	!Speeds
	CONST speeddata WorkingstepSpeeddatas{140} := [
		[ 800, 500, 5000, 1000],
		[ 800, 500, 5000, 1000],
		[ 4.23333333333333, 500, 5000, 1000],
		[ 4.23333333333333, 500, 5000, 1000],
		[ 800, 500, 5000, 1000],
		[ 800, 500, 5000, 1000],
		[ 800, 500, 5000, 1000],
		[ 800, 500, 5000, 1000],
		[ 800, 500, 5000, 1000],
		[ 4.23333333333333, 500, 5000, 1000],
		[ 4.23333333333333, 500, 5000, 1000],
		[ 800, 500, 5000, 1000],
		[ 800, 500, 5000, 1000],
		[ 800, 500, 5000, 1000],
		[ 800, 500, 5000, 1000],
		[ 800, 500, 5000, 1000],
		[ 4.23333333333333, 500, 5000, 1000],
		[ 4.23333333333333, 500, 5000, 1000],
		[ 800, 500, 5000, 1000],
		[ 800, 500, 5000, 1000],
		[ 800, 500, 5000, 1000],
		[ 800, 500, 5000, 1000],
		[ 800, 500, 5000, 1000],
		[ 4.23333333333333, 500, 5000, 1000],
		[ 4.23333333333333, 500, 5000, 1000],
		[ 800, 500, 5000, 1000],
		[ 800, 500, 5000, 1000],
		[ 800, 500, 5000, 1000],
		[ 800, 500, 5000, 1000],
		[ 800, 500, 5000, 1000],
		[ 4.23333333333333, 500, 5000, 1000],
		[ 4.23333333333333, 500, 5000, 1000],
		[ 800, 500, 5000, 1000],
		[ 800, 500, 5000, 1000],
		[ 800, 500, 5000, 1000],
		[ 800, 500, 5000, 1000],
		[ 800, 500, 5000, 1000],
		[ 4.23333333333333, 500, 5000, 1000],
		[ 4.23333333333333, 500, 5000, 1000],
		[ 800, 500, 5000, 1000],
		[ 800, 500, 5000, 1000],
		[ 800, 500, 5000, 1000],
		[ 800, 500, 5000, 1000],
		[ 800, 500, 5000, 1000],
		[ 4.23333333333333, 500, 5000, 1000],
		[ 4.23333333333333, 500, 5000, 1000],
		[ 800, 500, 5000, 1000],
		[ 800, 500, 5000, 1000],
		[ 800, 500, 5000, 1000],
		[ 800, 500, 5000, 1000],
		[ 800, 500, 5000, 1000],
		[ 4.23333333333333, 500, 5000, 1000],
		[ 4.23333333333333, 500, 5000, 1000],
		[ 800, 500, 5000, 1000],
		[ 800, 500, 5000, 1000],
		[ 800, 500, 5000, 1000],
		[ 800, 500, 5000, 1000],
		[ 800, 500, 5000, 1000],
		[ 4.23333333333333, 500, 5000, 1000],
		[ 4.23333333333333, 500, 5000, 1000],
		[ 800, 500, 5000, 1000],
		[ 800, 500, 5000, 1000],
		[ 800, 500, 5000, 1000],
		[ 800, 500, 5000, 1000],
		[ 800, 500, 5000, 1000],
		[ 4.23333333333333, 500, 5000, 1000],
		[ 4.23333333333333, 500, 5000, 1000],
		[ 800, 500, 5000, 1000],
		[ 800, 500, 5000, 1000],
		[ 800, 500, 5000, 1000],
		[ 800, 500, 5000, 1000],
		[ 800, 500, 5000, 1000],
		[ 4.23333333333333, 500, 5000, 1000],
		[ 4.23333333333333, 500, 5000, 1000],
		[ 800, 500, 5000, 1000],
		[ 800, 500, 5000, 1000],
		[ 800, 500, 5000, 1000],
		[ 800, 500, 5000, 1000],
		[ 800, 500, 5000, 1000],
		[ 4.23333333333333, 500, 5000, 1000],
		[ 4.23333333333333, 500, 5000, 1000],
		[ 800, 500, 5000, 1000],
		[ 800, 500, 5000, 1000],
		[ 800, 500, 5000, 1000],
		[ 800, 500, 5000, 1000],
		[ 800, 500, 5000, 1000],
		[ 4.23333333333333, 500, 5000, 1000],
		[ 4.23333333333333, 500, 5000, 1000],
		[ 800, 500, 5000, 1000],
		[ 800, 500, 5000, 1000],
		[ 800, 500, 5000, 1000],
		[ 800, 500, 5000, 1000],
		[ 800, 500, 5000, 1000],
		[ 4.23333333333333, 500, 5000, 1000],
		[ 4.23333333333333, 500, 5000, 1000],
		[ 800, 500, 5000, 1000],
		[ 800, 500, 5000, 1000],
		[ 800, 500, 5000, 1000],
		[ 800, 500, 5000, 1000],
		[ 800, 500, 5000, 1000],
		[ 4.23333333333333, 500, 5000, 1000],
		[ 4.23333333333333, 500, 5000, 1000],
		[ 800, 500, 5000, 1000],
		[ 800, 500, 5000, 1000],
		[ 800, 500, 5000, 1000],
		[ 800, 500, 5000, 1000],
		[ 800, 500, 5000, 1000],
		[ 4.23333333333333, 500, 5000, 1000],
		[ 4.23333333333333, 500, 5000, 1000],
		[ 800, 500, 5000, 1000],
		[ 800, 500, 5000, 1000],
		[ 800, 500, 5000, 1000],
		[ 800, 500, 5000, 1000],
		[ 800, 500, 5000, 1000],
		[ 4.23333333333333, 500, 5000, 1000],
		[ 4.23333333333333, 500, 5000, 1000],
		[ 800, 500, 5000, 1000],
		[ 800, 500, 5000, 1000],
		[ 800, 500, 5000, 1000],
		[ 800, 500, 5000, 1000],
		[ 800, 500, 5000, 1000],
		[ 4.23333333333333, 500, 5000, 1000],
		[ 4.23333333333333, 500, 5000, 1000],
		[ 800, 500, 5000, 1000],
		[ 800, 500, 5000, 1000],
		[ 800, 500, 5000, 1000],
		[ 800, 500, 5000, 1000],
		[ 800, 500, 5000, 1000],
		[ 4.23333333333333, 500, 5000, 1000],
		[ 4.23333333333333, 500, 5000, 1000],
		[ 800, 500, 5000, 1000],
		[ 800, 500, 5000, 1000],
		[ 800, 500, 5000, 1000],
		[ 800, 500, 5000, 1000],
		[ 800, 500, 5000, 1000],
		[ 4.23333333333333, 500, 5000, 1000],
		[ 4.23333333333333, 500, 5000, 1000],
		[ 800, 500, 5000, 1000],
		[ 800, 500, 5000, 1000],
		[ 800, 500, 5000, 1000]
		];


ENDMODULE

--- Backups/Rob2/RAPID/TASK1/PROGMOD/KyleWorkingPlan.mod ---
MODULE KyleWorkingPlan
  PERS string workingPlanUUID:="sdvonvskvnwovewn342532nkfloencvosnvqwef12";
    PERS string AP238_WORKINGSTEP_NAME := "";
    PERS string AP238_WORKINGSTEP_UUID := "";
    PERS string AP238_FEATURE_NAME := "";
    PERS string AP238_FEATURE_UUID := "";
    PERS bool ok;
    PERS num startIndex :=134;
    PERS num stopIndex :=140;
      CONST speeddata serge := [ 800, 500, 5000, 1000];



    PROC main()

       !  SetDO IsDone,0;
         MoveAbsJ jHome,v400,z10,PendEff_point\WObj:=A;
        MoveAbsJ jee,v400,z10,PendEff_point\WObj:=A;
        ConfJ\Off;
        ConfL\Off;

       FOR i FROM 1 TO dim(WorkPlan,1) DO

           ok := StrToVal(Workplan{i,1}, startIndex);
           ok := StrToVal(Workplan{i,2}, stopIndex);

                WorkingStep startIndex, stopIndex, Workplan{i,3}, Workplan{i,4}, Workplan{i,5}, Workplan{i,6}, WorkingstepRobtargets, WorkingstepSpeeddatas;

        ENDFOR

        MoveAbsJ jee,v400,z10,PendEff_point\WObj:=A;
        MoveAbsJ jHome,v400,z10,PendEff_point\WObj:=A;
        !SetDO IsDone,0;
    ENDPROC

    PROC WorkingStep(num startpos, num endpos, string workingstepName, string workingstepUUID, string featureName, string featureUUID, robtarget targetList{*}, speeddata speedList{*})

        FOR i FROM startpos TO endpos DO
      !           SetDO IsDone,0;
            AP238_WORKINGSTEP_NAME := workingstepName;
            AP238_WORKINGSTEP_UUID := workingstepUUID;
            AP238_FEATURE_NAME := featureName;
            AP238_FEATURE_UUID := featureUUID;
     !       MoveL targetList{i},v1000,z100,PendEff_point\WObj:=A;
            MoveL Workingsteprobtargets{i}, speedList{i}, z100,PendEff_point\WObj:=A;
     !       SetDO IsDone,1;
            AP238_WORKINGSTEP_NAME := "";
            AP238_WORKINGSTEP_UUID := "";
            AP238_FEATURE_NAME := "";
            AP238_FEATURE_UUID := "";
        ENDFOR

    ENDPROC

ENDMODULE

--- Backups/Rob2/RAPID/TASK1/SYSMOD/StandardJointMoves.sys ---
MODULE StandardJointMoves(SYSMODULE)
    !Home Joint Target
    CONST jointtarget jHome:=[[0,0,0,0,0,0],[9E+09,9E+09,9E+09,9E+09,9E+09,9E+09]];
    !Entry/Exit Joint Targets
    CONST jointtarget jee:=[[90,14,18,4,-38,0],[9E+09,9E+09,9E+09,9E+09,9E+09,9E+09]];
ENDMODULE

--- Backups/Rob2/RAPID/TASK1/SYSMOD/WorkObjs.sys ---
MODULE WorkObjs(SYSMODULE)
   TASK PERS wobjdata A:=[FALSE,TRUE,"",[[246.014,597.3,290.101],[0,0,0,1]],[[0,0,0],[1,0,0,0]]];
ENDMODULE

--- Backups/Rob3/RAPID/TASK1/PROGMOD/CartmanTargets.mod ---
MODULE CartmanTargets

	!Workplan Variables
	CONST string workplanName := "Cartman";
	CONST string workplanUUID := "e8924aac-08a1-45c9-8646-5367342a41b0";

	!Workingsteps
	CONST string WorkPlan{20,6} := [
		["1","7", "Drilling.82", "d2e6eab3-8d0a-4f0f-a95d-911cd3530854", "Hole.182", "99ddfef0-3deb-445b-9c3c-e9123ea0c45e"],
		["8","14", "Drilling.77", "18dec0f3-9a71-4d62-9ffd-4b071a4c2c96", "Hole.187", "ac14d56a-bac8-4703-abe8-8083d949a042"],
		["15","21", "Drilling.77A", "cce52ede-30b0-41b1-9812-f49428268d42", "Hole.186", "13f6412f-3d62-4080-9683-c1b012cf2329"],
		["22","28", "Drilling.81", "cc8ebbb7-3856-4b1d-89e7-3bb7927c75a5", "Hole.183", "cc7cadc1-0fbf-4952-a172-cb43c9784d58"],
		["29","35", "Drilling.82A", "fb1fd053-2caa-42bb-a221-a69a247b4566", "Hole.181", "d6ab53ed-32cb-4e94-b962-5e5bce2dd949"],
		["36","42", "Drilling.78", "0ce5bf9a-dc56-429d-9ede-9ff3cf936782", "Hole.188", "61b61ac0-b937-4570-af27-f3e5565ecb41"],
		["43","49", "Drilling.80", "097974f7-0281-41d6-be47-a718a708f2c1", "Hole.184", "41873095-e461-4717-85b4-deda62e7cc48"],
		["50","56", "Drilling.79", "0d38a1e5-c414-47eb-bffd-0c035c73e724", "Hole.189", "7aab888b-ee1b-4aa6-95a1-195311f5c09c"],
		["57","63", "Drilling.56", "71fb19fa-6caa-4311-b6e3-cc7c1a002d0e", "Hole.193", "534c8ca5-8759-4bfe-8b3a-f64014fb1b37"],
		["64","70", "Drilling.57", "82dc275d-79a1-4817-aca9-f89dbea4337b", "Hole.194", "b7011f38-5032-4673-a101-1254335b2b68"],
		["71","77", "Drilling.58", "e8ffa874-f10e-4ad9-b179-7e628cd38fb4", "Hole.195", "b2305f3a-4977-4727-8945-7fbced9dd981"],
		["78","84", "Drilling.59", "0436a6f4-bfce-4d24-b9fc-4974d9771220", "Hole.196", "3f2baa8f-1c3f-4c1c-9c8e-c6857731bbd6"],
		["85","91", "Drilling.60", "c922b515-5149-48e0-b3c2-25974a63925d", "Hole.199", "9f4fe053-f702-4970-bd3b-e9d6d5939926"],
		["92","98", "Drilling.61", "54f7aa6c-4c3b-4a01-975b-a374c0101e01", "Hole.198", "0cbf5231-fc2b-4c71-8eca-d485859f5bef"],
		["99","105", "Drilling.62", "308c7519-319c-495b-866e-887c108f69fd", "Hole.197", "97270ee4-7d12-42d9-b2be-af7000f13095"],
		["106","112", "Drilling.63", "ae041463-52c1-413a-bc8f-b82ceccd6cbf", "Hole.192", "a8675cfd-087c-4d76-9144-1d9942c5b76b"],
		["113","119", "Drilling.96", "366ca4c1-51ca-4762-a30e-71a9ecae8757", "Hole.176", "5d7c72e5-ba80-4f5c-9be4-85262b61495c"],
		["120","126", "Drilling.97", "81b03597-23b4-45f9-8253-620e9a46ff2e", "Hole.177", "fbc5cc65-6031-4a9a-8bf6-0c8b0c46d944"],
		["127","133", "Drilling.98", "d04a2e7a-5080-477a-8967-be3c7ad103b0", "Hole.178", "14004e87-3834-406b-b1c2-5711ea87ae56"],
		["134","140", "Drilling.99", "80c84945-9521-4e27-bda3-a7734aa46377", "Hole.179", "ec45e44e-466b-44fe-87e7-d5d7371b5502"]
		];

	!Positions
	CONST robtarget WorkingstepRobtargets{140} := [
		[[1250.47999638542,-108.227438181067,34.9975797061398],[0.00721600922388558,-0.000419915796535777,-0.998285039502953,-0.0580924503373097],[0,0,0,0],[9E+09,9E+09,9E+09,9E+09,9E+09,9E+09]],
		[[1249.75058558968,-102.335059394747,-15.4542570506085],[0.00721600922388558,-0.000419915796535777,-0.998285039502953,-0.0580924503373097],[0,0,0,0],[9E+09,9E+09,9E+09,9E+09,9E+09,9E+09]],
		[[1249.75058558968,-102.335059394747,-15.4542570506085],[0.00721600922388558,-0.000419915796535777,-0.998285039502953,-0.0580924503373097],[0,0,0,0],[9E+09,9E+09,9E+09,9E+09,9E+09,9E+09]],
		[[1249.29470384234,-98.6523226532974,-46.9866550235762],[0.00721600922388558,-0.000419915796535777,-0.998285039502953,-0.0580924503373097],[0,0,0,0],[9E+09,9E+09,9E+09,9E+09,9E+09,9E+09]],
		[[1249.29470384234,-98.6523226532974,-46.9866550235762],[0.00721600922388558,-0.000419915796535777,-0.998285039502953,-0.0580924503373097],[0,0,0,0],[9E+09,9E+09,9E+09,9E+09,9E+09,9E+09]],
		[[1249.75058558968,-102.335059394747,-15.4542570506085],[0.00721600922388558,-0.000419915796535777,-0.998285039502953,-0.0580924503373097],[0,0,0,0],[9E+09,9E+09,9E+09,9E+09,9E+09,9E+09]],
		[[1250.47999638542,-108.227438181067,34.9975797061398],[0.00721600922388558,-0.000419915796535777,-0.998285039502953,-0.0580924503373097],[0,0,0,0],[9E+09,9E+09,9E+09,9E+09,9E+09,9E+09]],
		[[1190.4996392186,-113.751032090431,35.2122877951345],[0.00727717079532053,-0.000437833858996109,-0.998168434785264,-0.0600551986514469],[0,0,0,0],[9E+09,9E+09,9E+09,9E+09,9E+09,9E+09]],
		[[1189.76430434352,-107.660275683661,-15.2158984603209],[0.00727717079532053,-0.000437833858996109,-0.998168434785264,-0.0600551986514469],[0,0,0,0],[9E+09,9E+09,9E+09,9E+09,9E+09,9E+09]],
		[[1189.76430434352,-107.660275683661,-15.2158984603209],[0.00727717079532053,-0.000437833858996109,-0.998168434785264,-0.0600551986514469],[0,0,0,0],[9E+09,9E+09,9E+09,9E+09,9E+09,9E+09]],
		[[1189.3047200466,-103.853552929431,-46.7335148699807],[0.00727717079532053,-0.000437833858996109,-0.998168434785264,-0.0600551986514469],[0,0,0,0],[9E+09,9E+09,9E+09,9E+09,9E+09,9E+09]],
		[[1189.3047200466,-103.853552929431,-46.7335148699807],[0.00727717079532053,-0.000437833858996109,-0.998168434785264,-0.0600551986514469],[0,0,0,0],[9E+09,9E+09,9E+09,9E+09,9E+09,9E+09]],
		[[1189.76430434352,-107.660275683661,-15.2158984603209],[0.00727717079532053,-0.000437833858996109,-0.998168434785264,-0.0600551986514469],[0,0,0,0],[9E+09,9E+09,9E+09,9E+09,9E+09,9E+09]],
		[[1190.4996392186,-113.751032090431,35.2122877951345],[0.00727717079532053,-0.000437833858996109,-0.998168434785264,-0.0600551986514469],[0,0,0,0],[9E+09,9E+09,9E+09,9E+09,9E+09,9E+09]],
		[[1189.80854349765,-65.9236756789968,39.7730886825223],[0.00665335945126355,-0.000231418506074151,-0.999373500218657,-0.0347604130326124],[0,0,0,0],[9E+09,9E+09,9E+09,9E+09,9E+09,9E+09]],
		[[1189.13380297056,-62.3940738632379,-10.8996518812492],[0.00665335945126355,-0.000231418506074151,-0.999373500218657,-0.0347604130326124],[0,0,0,0],[9E+09,9E+09,9E+09,9E+09,9E+09,9E+09]],
		[[1189.13380297056,-62.3940738632379,-10.8996518812492],[0.00665335945126355,-0.000231418506074151,-0.999373500218657,-0.0347604130326124],[0,0,0,0],[9E+09,9E+09,9E+09,9E+09,9E+09,9E+09]],
		[[1188.71209014113,-60.1880727283885,-42.5701147336066],[0.00665335945126355,-0.000231418506074151,-0.999373500218657,-0.0347604130326124],[0,0,0,0],[9E+09,9E+09,9E+09,9E+09,9E+09,9E+09]],
		[[1188.71209014113,-60.1880727283885,-42.5701147336066],[0.00665335945126355,-0.000231418506074151,-0.999373500218657,-0.0347604130326124],[0,0,0,0],[9E+09,9E+09,9E+09,9E+09,9E+09,9E+09]],
		[[1189.13380297056,-62.3940738632379,-10.8996518812492],[0.00665335945126355,-0.000231418506074151,-0.999373500218657,-0.0347604130326124],[0,0,0,0],[9E+09,9E+09,9E+09,9E+09,9E+09,9E+09]],
		[[1189.80854349765,-65.9236756789968,39.7730886825223],[0.00665335945126355,-0.000231418506074151,-0.999373500218657,-0.0347604130326124],[0,0,0,0],[9E+09,9E+09,9E+09,9E+09,9E+09,9E+09]],
		[[1251.74376412468,-153.597058265429,28.5448951127816],[0.00812040995990566,-0.000673216620954281,-0.996547971260864,-0.0826180773034575],[0,0,0,0],[9E+09,9E+09,9E+09,9E+09,9E+09,9E+09]],
		[[1250.92722949069,-145.231482502716,-21.5549094112862],[0.00812040995990566,-0.000673216620954281,-0.996547971260864,-0.0826180773034575],[0,0,0,0],[9E+09,9E+09,9E+09,9E+09,9E+09,9E+09]],
		[[1250.92722949069,-145.231482502716,-21.5549094112862],[0.00812040995990566,-0.000673216620954281,-0.996547971260864,-0.0826180773034575],[0,0,0,0],[9E+09,9E+09,9E+09,9E+09,9E+09,9E+09]],
		[[1250.41689534445,-140.002997651021,-52.8672872388287],[0.00812040995990566,-0.000673216620954281,-0.996547971260864,-0.0826180773034575],[0,0,0,0],[9E+09,9E+09,9E+09,9E+09,9E+09,9E+09]],
		[[1250.41689534445,-140.002997651021,-52.8672872388287],[0.00812040995990566,-0.000673216620954281,-0.996547971260864,-0.0826180773034575],[0,0,0,0],[9E+09,9E+09,9E+09,9E+09,9E+09,9E+09]],
		[[1250.92722949069,-145.231482502716,-21.5549094112862],[0.00812040995990566,-0.000673216620954281,-0.996547971260864,-0.0826180773034575],[0,0,0,0],[9E+09,9E+09,9E+09,9E+09,9E+09,9E+09]],
		[[1251.74376412468,-153.597058265429,28.5448951127816],[0.00812040995990566,-0.000673216620954281,-0.996547971260864,-0.0826180773034575],[0,0,0,0],[9E+09,9E+09,9E+09,9E+09,9E+09,9E+09]],
		[[1251.30388547251,-68.6381103493351,38.7572467507825],[0.0066912868110706,-0.000246540181525224,-0.99929951275717,-0.0368191485783281],[0,0,0,0],[9E+09,9E+09,9E+09,9E+09,9E+09,9E+09]],
		[[1250.62544921187,-64.8997376477342,-11.9004702702614],[0.0066912868110706,-0.000246540181525224,-0.99929951275717,-0.0368191485783281],[0,0,0,0],[9E+09,9E+09,9E+09,9E+09,9E+09,9E+09]],
		[[1250.62544921187,-64.8997376477342,-11.9004702702614],[0.0066912868110706,-0.000246540181525224,-0.99929951275717,-0.0368191485783281],[0,0,0,0],[9E+09,9E+09,9E+09,9E+09,9E+09,9E+09]],
		[[1250.20142654896,-62.5632547092337,-43.5615434084138],[0.0066912868110706,-0.000246540181525224,-0.99929951275717,-0.0368191485783281],[0,0,0,0],[9E+09,9E+09,9E+09,9E+09,9E+09,9E+09]],
		[[1250.20142654896,-62.5632547092337,-43.5615434084138],[0.0066912868110706,-0.000246540181525224,-0.99929951275717,-0.0368191485783281],[0,0,0,0],[9E+09,9E+09,9E+09,9E+09,9E+09,9E+09]],
		[[1250.62544921187,-64.8997376477342,-11.9004702702614],[0.0066912868110706,-0.000246540181525224,-0.99929951275717,-0.0368191485783281],[0,0,0,0],[9E+09,9E+09,9E+09,9E+09,9E+09,9E+09]],
		[[1251.30388547251,-68.6381103493351,38.7572467507825],[0.0066912868110706,-0.000246540181525224,-0.99929951275717,-0.0368191485783281],[0,0,0,0],[9E+09,9E+09,9E+09,9E+09,9E+09,9E+09]],
		[[1190.60083196625,-155.158216713176,29.2801865539037],[0.00809702025081855,-0.000666620341839099,-0.996595199463999,-0.0820487799159123],[0,0,0,0],[9E+09,9E+09,9E+09,9E+09,9E+09,9E+09]],
		[[1189.78653274383,-146.849895222209,-20.8291809413968],[0.00809702025081855,-0.000666620341839099,-0.996595199463999,-0.0820487799159123],[0,0,0,0],[9E+09,9E+09,9E+09,9E+09,9E+09,9E+09]],
		[[1189.78653274383,-146.849895222209,-20.8291809413968],[0.00809702025081855,-0.000666620341839099,-0.996595199463999,-0.0820487799159123],[0,0,0,0],[9E+09,9E+09,9E+09,9E+09,9E+09,9E+09]],
		[[1189.27759572982,-141.657194290354,-52.1475356259597],[0.00809702025081855,-0.000666620341839099,-0.996595199463999,-0.0820487799159123],[0,0,0,0],[9E+09,9E+09,9E+09,9E+09,9E+09,9E+09]],
		[[1189.27759572982,-141.657194290354,-52.1475356259597],[0.00809702025081855,-0.000666620341839099,-0.996595199463999,-0.0820487799159123],[0,0,0,0],[9E+09,9E+09,9E+09,9E+09,9E+09,9E+09]],
		[[1189.78653274383,-146.849895222209,-20.8291809413968],[0.00809702025081855,-0.000666620341839099,-0.996595199463999,-0.0820487799159123],[0,0,0,0],[9E+09,9E+09,9E+09,9E+09,9E+09,9E+09]],
		[[1190.60083196625,-155.158216713176,29.2801865539037],[0.00809702025081855,-0.000666620341839099,-0.996595199463999,-0.0820487799159123],[0,0,0,0],[9E+09,9E+09,9E+09,9E+09,9E+09,9E+09]],
		[[1251.64830610495,-198.940144194599,19.8167872449908],[0.00936178502431022,-0.00100991908065343,-0.99418752340432,-0.107249733574467],[0,0,0,0],[9E+09,9E+09,9E+09,9E+09,9E+09,9E+09]],
		[[1250.71368198328,-188.105946746604,-29.8056536805528],[0.00936178502431022,-0.00100991908065343,-0.99418752340432,-0.107249733574467],[0,0,0,0],[9E+09,9E+09,9E+09,9E+09,9E+09,9E+09]],
		[[1250.71368198328,-188.105946746604,-29.8056536805528],[0.00936178502431022,-0.00100991908065343,-0.99418752340432,-0.107249733574467],[0,0,0,0],[9E+09,9E+09,9E+09,9E+09,9E+09,9E+09]],
		[[1250.12954190724,-181.334573341607,-60.8196792590172],[0.00936178502431022,-0.00100991908065343,-0.99418752340432,-0.107249733574467],[0,0,0,0],[9E+09,9E+09,9E+09,9E+09,9E+09,9E+09]],
		[[1250.12954190724,-181.334573341607,-60.8196792590172],[0.00936178502431022,-0.00100991908065343,-0.99418752340432,-0.107249733574467],[0,0,0,0],[9E+09,9E+09,9E+09,9E+09,9E+09,9E+09]],
		[[1250.71368198328,-188.105946746604,-29.8056536805528],[0.00936178502431022,-0.00100991908065343,-0.99418752340432,-0.107249733574467],[0,0,0,0],[9E+09,9E+09,9E+09,9E+09,9E+09,9E+09]],
		[[1251.64830610495,-198.940144194599,19.8167872449908],[0.00936178502431022,-0.00100991908065343,-0.99418752340432,-0.107249733574467],[0,0,0,0],[9E+09,9E+09,9E+09,9E+09,9E+09,9E+09]],
		[[1191.95221981654,-205.961103975954,19.400651812078],[0.00947883770226787,-0.00104166552827841,-0.99397062768479,-0.109231212886453],[0,0,0,0],[9E+09,9E+09,9E+09,9E+09,9E+09,9E+09]],
		[[1191.00653678319,-194.929122888932,-30.1779834746662],[0.00947883770226787,-0.00104166552827841,-0.99397062768479,-0.109231212886453],[0,0,0,0],[9E+09,9E+09,9E+09,9E+09,9E+09,9E+09]],
		[[1191.00653678319,-194.929122888932,-30.1779834746662],[0.00947883770226787,-0.00104166552827841,-0.99397062768479,-0.109231212886453],[0,0,0,0],[9E+09,9E+09,9E+09,9E+09,9E+09,9E+09]],
		[[1190.41548488734,-188.034134709543,-61.1646305288814],[0.00947883770226787,-0.00104166552827841,-0.99397062768479,-0.109231212886453],[0,0,0,0],[9E+09,9E+09,9E+09,9E+09,9E+09,9E+09]],
		[[1190.41548488734,-188.034134709543,-61.1646305288814],[0.00947883770226787,-0.00104166552827841,-0.99397062768479,-0.109231212886453],[0,0,0,0],[9E+09,9E+09,9E+09,9E+09,9E+09,9E+09]],
		[[1191.00653678319,-194.929122888932,-30.1779834746662],[0.00947883770226787,-0.00104166552827841,-0.99397062768479,-0.109231212886453],[0,0,0,0],[9E+09,9E+09,9E+09,9E+09,9E+09,9E+09]],
		[[1191.95221981654,-205.961103975954,19.400651812078],[0.00947883770226787,-0.00104166552827841,-0.99397062768479,-0.109231212886453],[0,0,0,0],[9E+09,9E+09,9E+09,9E+09,9E+09,9E+09]],
		[[1047.46148935396,-72.0531501973382,41.2352412437369],[0.00668721181442413,-0.000244662737514811,-0.999309004762805,-0.0365613776855514],[0,0,0,0],[9E+09,9E+09,9E+09,9E+09,9E+09,9E+09]],
		[[1046.7834469431,-68.3409147913177,-9.42440311722726],[0.00668721181442413,-0.000244662737514811,-0.999309004762805,-0.0365613776855514],[0,0,0,0],[9E+09,9E+09,9E+09,9E+09,9E+09,9E+09]],
		[[1046.7834469431,-68.3409147913177,-9.42440311722726],[0.00668721181442413,-0.000244662737514811,-0.999309004762805,-0.0365613776855514],[0,0,0,0],[9E+09,9E+09,9E+09,9E+09,9E+09,9E+09]],
		[[1046.35967043631,-66.0207676625549,-41.0866808428298],[0.00668721181442413,-0.000244662737514811,-0.999309004762805,-0.0365613776855514],[0,0,0,0],[9E+09,9E+09,9E+09,9E+09,9E+09,9E+09]],
		[[1046.35967043631,-66.0207676625549,-41.0866808428298],[0.00668721181442413,-0.000244662737514811,-0.999309004762805,-0.0365613776855514],[0,0,0,0],[9E+09,9E+09,9E+09,9E+09,9E+09,9E+09]],
		[[1046.7834469431,-68.3409147913177,-9.42440311722726],[0.00668721181442413,-0.000244662737514811,-0.999309004762805,-0.0365613776855514],[0,0,0,0],[9E+09,9E+09,9E+09,9E+09,9E+09,9E+09]],
		[[1047.46148935396,-72.0531501973382,41.2352412437369],[0.00668721181442413,-0.000244662737514811,-0.999309004762805,-0.0365613776855514],[0,0,0,0],[9E+09,9E+09,9E+09,9E+09,9E+09,9E+09]],
		[[1052.42343074024,-109.067908351377,37.7494232893189],[0.00713988796543304,-0.000396579657530434,-0.998435450217324,-0.0554573392234659],[0,0,0,0],[9E+09,9E+09,9E+09,9E+09,9E+09,9E+09]],
		[[1051.70138758157,-103.441970404417,-12.7329248721323],[0.00713988796543304,-0.000396579657530434,-0.998435450217324,-0.0554573392234659],[0,0,0,0],[9E+09,9E+09,9E+09,9E+09,9E+09,9E+09]],
		[[1051.70138758157,-103.441970404417,-12.7329248721323],[0.00713988796543304,-0.000396579657530434,-0.998435450217324,-0.0554573392234659],[0,0,0,0],[9E+09,9E+09,9E+09,9E+09,9E+09,9E+09]],
		[[1051.2501106074,-99.9257591875673,-44.2843924730394],[0.00713988796543304,-0.000396579657530434,-0.998435450217324,-0.0554573392234659],[0,0,0,0],[9E+09,9E+09,9E+09,9E+09,9E+09,9E+09]],
		[[1051.2501106074,-99.9257591875673,-44.2843924730394],[0.00713988796543304,-0.000396579657530434,-0.998435450217324,-0.0554573392234659],[0,0,0,0],[9E+09,9E+09,9E+09,9E+09,9E+09,9E+09]],
		[[1051.70138758157,-103.441970404417,-12.7329248721323],[0.00713988796543304,-0.000396579657530434,-0.998435450217324,-0.0554573392234659],[0,0,0,0],[9E+09,9E+09,9E+09,9E+09,9E+09,9E+09]],
		[[1052.42343074024,-109.067908351377,37.7494232893189],[0.00713988796543304,-0.000396579657530434,-0.998435450217324,-0.0554573392234659],[0,0,0,0],[9E+09,9E+09,9E+09,9E+09,9E+09,9E+09]],
		[[1058.4740893206,-161.105031430509,30.4416121484464],[0.00810621924312884,-0.000668612028545384,-0.996582703082117,-0.0821995017325489],[0,0,0,0],[9E+09,9E+09,9E+09,9E+09,9E+09,9E+09]],
		[[1057.65889579635,-152.781550841607,-19.6652250138031],[0.00810621924312884,-0.000668612028545384,-0.996582703082117,-0.0821995017325489],[0,0,0,0],[9E+09,9E+09,9E+09,9E+09,9E+09,9E+09]],
		[[1057.65889579635,-152.781550841607,-19.6652250138031],[0.00810621924312884,-0.000668612028545384,-0.996582703082117,-0.0821995017325489],[0,0,0,0],[9E+09,9E+09,9E+09,9E+09,9E+09,9E+09]],
		[[1057.1493998437,-147.579375473542,-50.981998240209],[0.00810621924312884,-0.000668612028545384,-0.996582703082117,-0.0821995017325489],[0,0,0,0],[9E+09,9E+09,9E+09,9E+09,9E+09,9E+09]],
		[[1057.1493998437,-147.579375473542,-50.981998240209],[0.00810621924312884,-0.000668612028545384,-0.996582703082117,-0.0821995017325489],[0,0,0,0],[9E+09,9E+09,9E+09,9E+09,9E+09,9E+09]],
		[[1057.65889579635,-152.781550841607,-19.6652250138031],[0.00810621924312884,-0.000668612028545384,-0.996582703082117,-0.0821995017325489],[0,0,0,0],[9E+09,9E+09,9E+09,9E+09,9E+09,9E+09]],
		[[1058.4740893206,-161.105031430509,30.4416121484464],[0.00810621924312884,-0.000668612028545384,-0.996582703082117,-0.0821995017325489],[0,0,0,0],[9E+09,9E+09,9E+09,9E+09,9E+09,9E+09]],
		[[1057.93506911126,-221.171435306608,18.5414921384049],[0.00971864696644204,-0.00110695702979796,-0.993528265759436,-0.113163190500817],[0,0,0,0],[9E+09,9E+09,9E+09,9E+09,9E+09,9E+09]],
		[[1056.96677196969,-209.747370115093,-30.9478313076238],[0.00971864696644204,-0.00110695702979796,-0.993528265759436,-0.113163190500817],[0,0,0,0],[9E+09,9E+09,9E+09,9E+09,9E+09,9E+09]],
		[[1056.96677196969,-209.747370115093,-30.9478313076238],[0.00971864696644204,-0.00110695702979796,-0.993528265759436,-0.113163190500817],[0,0,0,0],[9E+09,9E+09,9E+09,9E+09,9E+09,9E+09]],
		[[1056.36158625621,-202.607329370396,-61.8786584613916],[0.00971864696644204,-0.00110695702979796,-0.993528265759436,-0.113163190500817],[0,0,0,0],[9E+09,9E+09,9E+09,9E+09,9E+09,9E+09]],
		[[1056.36158625621,-202.607329370396,-61.8786584613916],[0.00971864696644204,-0.00110695702979796,-0.993528265759436,-0.113163190500817],[0,0,0,0],[9E+09,9E+09,9E+09,9E+09,9E+09,9E+09]],
		[[1056.96677196969,-209.747370115093,-30.9478313076238],[0.00971864696644204,-0.00110695702979796,-0.993528265759436,-0.113163190500817],[0,0,0,0],[9E+09,9E+09,9E+09,9E+09,9E+09,9E+09]],
		[[1057.93506911126,-221.171435306608,18.5414921384049],[0.00971864696644204,-0.00110695702979796,-0.993528265759436,-0.113163190500817],[0,0,0,0],[9E+09,9E+09,9E+09,9E+09,9E+09,9E+09]],
		[[1127.85981856446,-218.635862664587,17.7574554971789],[0.00976696523800443,-0.0011207663604795,-0.993432439926763,-0.113997094585619],[0,0,0,0],[9E+09,9E+09,9E+09,9E+09,9E+09,9E+09]],
		[[1126.88699287504,-207.128711860815,-31.7125262145345],[0.00976696523800443,-0.0011207663604795,-0.993432439926763,-0.113997094585619],[0,0,0,0],[9E+09,9E+09,9E+09,9E+09,9E+09,9E+09]],
		[[1126.88699287504,-207.128711860815,-31.7125262145345],[0.00976696523800443,-0.0011207663604795,-0.993432439926763,-0.113997094585619],[0,0,0,0],[9E+09,9E+09,9E+09,9E+09,9E+09,9E+09]],
		[[1126.27897681915,-199.936742608458,-62.6312647843553],[0.00976696523800443,-0.0011207663604795,-0.993432439926763,-0.113997094585619],[0,0,0,0],[9E+09,9E+09,9E+09,9E+09,9E+09,9E+09]],
		[[1126.27897681915,-199.936742608458,-62.6312647843553],[0.00976696523800443,-0.0011207663604795,-0.993432439926763,-0.113997094585619],[0,0,0,0],[9E+09,9E+09,9E+09,9E+09,9E+09,9E+09]],
		[[1126.88699287504,-207.128711860815,-31.7125262145345],[0.00976696523800443,-0.0011207663604795,-0.993432439926763,-0.113997094585619],[0,0,0,0],[9E+09,9E+09,9E+09,9E+09,9E+09,9E+09]],
		[[1127.85981856446,-218.635862664587,17.7574554971789],[0.00976696523800443,-0.0011207663604795,-0.993432439926763,-0.113997094585619],[0,0,0,0],[9E+09,9E+09,9E+09,9E+09,9E+09,9E+09]],
		[[1128.43014953787,-163.53542979742,28.8839393142151],[0.00823029283472108,-0.000702478845333139,-0.996343236229819,-0.0850407221419141],[0,0,0,0],[9E+09,9E+09,9E+09,9E+09,9E+09,9E+09]],
		[[1127.60307907723,-154.926299957873,-21.1744150121005],[0.00823029283472108,-0.000702478845333139,-0.996343236229819,-0.0850407221419141],[0,0,0,0],[9E+09,9E+09,9E+09,9E+09,9E+09,9E+09]],
		[[1127.60307907723,-154.926299957873,-21.1744150121005],[0.00823029283472108,-0.000702478845333139,-0.996343236229819,-0.0850407221419141],[0,0,0,0],[9E+09,9E+09,9E+09,9E+09,9E+09,9E+09]],
		[[1127.08616003933,-149.545593808156,-52.4608864660477],[0.00823029283472108,-0.000702478845333139,-0.996343236229819,-0.0850407221419141],[0,0,0,0],[9E+09,9E+09,9E+09,9E+09,9E+09,9E+09]],
		[[1127.08616003933,-149.545593808156,-52.4608864660477],[0.00823029283472108,-0.000702478845333139,-0.996343236229819,-0.0850407221419141],[0,0,0,0],[9E+09,9E+09,9E+09,9E+09,9E+09,9E+09]],
		[[1127.60307907723,-154.926299957873,-21.1744150121005],[0.00823029283472108,-0.000702478845333139,-0.996343236229819,-0.0850407221419141],[0,0,0,0],[9E+09,9E+09,9E+09,9E+09,9E+09,9E+09]],
		[[1128.43014953787,-163.53542979742,28.8839393142151],[0.00823029283472108,-0.000702478845333139,-0.996343236229819,-0.0850407221419141],[0,0,0,0],[9E+09,9E+09,9E+09,9E+09,9E+09,9E+09]],
		[[1127.5520604083,-112.02129801337,36.3318839337975],[0.00721835054793264,-0.000420303654481913,-0.9982830037692,-0.0581271291717486],[0,0,0,0],[9E+09,9E+09,9E+09,9E+09,9E+09,9E+09]],
		[[1126.82241740506,-106.125413538039,-14.1195399047956],[0.00721835054793264,-0.000420303654481913,-0.9982830037692,-0.0581271291717486],[0,0,0,0],[9E+09,9E+09,9E+09,9E+09,9E+09,9E+09]],
		[[1126.82241740506,-106.125413538039,-14.1195399047956],[0.00721835054793264,-0.000420303654481913,-0.9982830037692,-0.0581271291717486],[0,0,0,0],[9E+09,9E+09,9E+09,9E+09,9E+09,9E+09]],
		[[1126.36639052804,-102.440485740957,-45.6516798039163],[0.00721835054793264,-0.000420303654481913,-0.9982830037692,-0.0581271291717486],[0,0,0,0],[9E+09,9E+09,9E+09,9E+09,9E+09,9E+09]],
		[[1126.36639052804,-102.440485740957,-45.6516798039163],[0.00721835054793264,-0.000420303654481913,-0.9982830037692,-0.0581271291717486],[0,0,0,0],[9E+09,9E+09,9E+09,9E+09,9E+09,9E+09]],
		[[1126.82241740506,-106.125413538039,-14.1195399047956],[0.00721835054793264,-0.000420303654481913,-0.9982830037692,-0.0581271291717486],[0,0,0,0],[9E+09,9E+09,9E+09,9E+09,9E+09,9E+09]],
		[[1127.5520604083,-112.02129801337,36.3318839337975],[0.00721835054793264,-0.000420303654481913,-0.9982830037692,-0.0581271291717486],[0,0,0,0],[9E+09,9E+09,9E+09,9E+09,9E+09,9E+09]],
		[[1128.61924471962,-66.6938481139753,40.5341707855242],[0.00665039597780486,-0.00023013398092707,-0.999379672280555,-0.0345830869660357],[0,0,0,0],[9E+09,9E+09,9E+09,9E+09,9E+09,9E+09]],
		[[1127.94479223978,-63.1822305905469,-10.1398230991262],[0.00665039597780486,-0.00023013398092707,-0.999379672280555,-0.0345830869660357],[0,0,0,0],[9E+09,9E+09,9E+09,9E+09,9E+09,9E+09]],
		[[1127.94479223978,-63.1822305905469,-10.1398230991262],[0.00665039597780486,-0.00023013398092707,-0.999379672280555,-0.0345830869660357],[0,0,0,0],[9E+09,9E+09,9E+09,9E+09,9E+09,9E+09]],
		[[1127.52325943989,-60.9874696384043,-41.811069277033],[0.00665039597780486,-0.00023013398092707,-0.999379672280555,-0.0345830869660357],[0,0,0,0],[9E+09,9E+09,9E+09,9E+09,9E+09,9E+09]],
		[[1127.52325943989,-60.9874696384043,-41.811069277033],[0.00665039597780486,-0.00023013398092707,-0.999379672280555,-0.0345830869660357],[0,0,0,0],[9E+09,9E+09,9E+09,9E+09,9E+09,9E+09]],
		[[1127.94479223978,-63.1822305905469,-10.1398230991262],[0.00665039597780486,-0.00023013398092707,-0.999379672280555,-0.0345830869660357],[0,0,0,0],[9E+09,9E+09,9E+09,9E+09,9E+09,9E+09]],
		[[1128.61924471962,-66.6938481139753,40.5341707855242],[0.00665039597780486,-0.00023013398092707,-0.999379672280555,-0.0345830869660357],[0,0,0,0],[9E+09,9E+09,9E+09,9E+09,9E+09,9E+09]],
		[[1280.40535998915,-77.4781676063704,37.6669469437901],[0.00679504073904094,-0.000285047734089657,-0.999098177542344,-0.0419115473433251],[0,0,0,0],[9E+09,9E+09,9E+09,9E+09,9E+09,9E+09]],
		[[1279.7168202408,-73.2235977584369,-12.9498936176672],[0.00679504073904094,-0.000285047734089657,-0.999098177542344,-0.0419115473433251],[0,0,0,0],[9E+09,9E+09,9E+09,9E+09,9E+09,9E+09]],
		[[1279.7168202408,-73.2235977584369,-12.9498936176672],[0.00679504073904094,-0.000285047734089657,-0.999098177542344,-0.0419115473433251],[0,0,0,0],[9E+09,9E+09,9E+09,9E+09,9E+09,9E+09]],
		[[1279.28648289808,-70.5644916034785,-44.5854189685778],[0.00679504073904094,-0.000285047734089657,-0.999098177542344,-0.0419115473433251],[0,0,0,0],[9E+09,9E+09,9E+09,9E+09,9E+09,9E+09]],
		[[1279.28648289808,-70.5644916034785,-44.5854189685778],[0.00679504073904094,-0.000285047734089657,-0.999098177542344,-0.0419115473433251],[0,0,0,0],[9E+09,9E+09,9E+09,9E+09,9E+09,9E+09]],
		[[1279.7168202408,-73.2235977584369,-12.9498936176672],[0.00679504073904094,-0.000285047734089657,-0.999098177542344,-0.0419115473433251],[0,0,0,0],[9E+09,9E+09,9E+09,9E+09,9E+09,9E+09]],
		[[1280.40535998915,-77.4781676063704,37.6669469437901],[0.00679504073904094,-0.000285047734089657,-0.999098177542344,-0.0419115473433251],[0,0,0,0],[9E+09,9E+09,9E+09,9E+09,9E+09,9E+09]],
		[[1277.40817693077,-117.472016129421,33.472734421395],[0.00738904055701226,-0.000470569704976723,-0.99795091498347,-0.0635543226496346],[0,0,0,0],[9E+09,9E+09,9E+09,9E+09,9E+09,9E+09]],
		[[1276.66202723732,-111.027774865225,-16.911340594068],[0.00738904055701226,-0.000470569704976723,-0.99795091498347,-0.0635543226496346],[0,0,0,0],[9E+09,9E+09,9E+09,9E+09,9E+09,9E+09]],
		[[1276.66202723732,-111.027774865225,-16.911340594068],[0.00738904055701226,-0.000470569704976723,-0.99795091498347,-0.0635543226496346],[0,0,0,0],[9E+09,9E+09,9E+09,9E+09,9E+09,9E+09]],
		[[1276.1956836789,-107.000124075103,-48.4013874787322],[0.00738904055701226,-0.000470569704976723,-0.99795091498347,-0.0635543226496346],[0,0,0,0],[9E+09,9E+09,9E+09,9E+09,9E+09,9E+09]],
		[[1276.1956836789,-107.000124075103,-48.4013874787322],[0.00738904055701226,-0.000470569704976723,-0.99795091498347,-0.0635543226496346],[0,0,0,0],[9E+09,9E+09,9E+09,9E+09,9E+09,9E+09]],
		[[1276.66202723732,-111.027774865225,-16.911340594068],[0.00738904055701226,-0.000470569704976723,-0.99795091498347,-0.0635543226496346],[0,0,0,0],[9E+09,9E+09,9E+09,9E+09,9E+09,9E+09]],
		[[1277.40817693077,-117.472016129421,33.472734421395],[0.00738904055701226,-0.000470569704976723,-0.99795091498347,-0.0635543226496346],[0,0,0,0],[9E+09,9E+09,9E+09,9E+09,9E+09,9E+09]],
		[[1277.64942637825,-158.123953639288,27.3488861055936],[0.00825634172421117,-0.000710159372976826,-0.996287002832898,-0.0856944366994647],[0,0,0,0],[9E+09,9E+09,9E+09,9E+09,9E+09,9E+09]],
		[[1276.81987972713,-149.449130570658,-22.6980848025598],[0.00825634172421117,-0.000710159372976826,-0.996287002832898,-0.0856944366994647],[0,0,0,0],[9E+09,9E+09,9E+09,9E+09,9E+09,9E+09]],
		[[1276.81987972713,-149.449130570658,-22.6980848025598],[0.00825634172421117,-0.000710159372976826,-0.996287002832898,-0.0856944366994647],[0,0,0,0],[9E+09,9E+09,9E+09,9E+09,9E+09,9E+09]],
		[[1276.30141307018,-144.027366152764,-53.9774416201559],[0.00825634172421117,-0.000710159372976826,-0.996287002832898,-0.0856944366994647],[0,0,0,0],[9E+09,9E+09,9E+09,9E+09,9E+09,9E+09]],
		[[1276.30141307018,-144.027366152764,-53.9774416201559],[0.00825634172421117,-0.000710159372976826,-0.996287002832898,-0.0856944366994647],[0,0,0,0],[9E+09,9E+09,9E+09,9E+09,9E+09,9E+09]],
		[[1276.81987972713,-149.449130570658,-22.6980848025598],[0.00825634172421117,-0.000710159372976826,-0.996287002832898,-0.0856944366994647],[0,0,0,0],[9E+09,9E+09,9E+09,9E+09,9E+09,9E+09]],
		[[1277.64942637825,-158.123953639288,27.3488861055936],[0.00825634172421117,-0.000710159372976826,-0.996287002832898,-0.0856944366994647],[0,0,0,0],[9E+09,9E+09,9E+09,9E+09,9E+09,9E+09]],
		[[1275.33381015192,-199.568058708582,19.231409467319],[0.00942251539533556,-0.00102672230604247,-0.994071031047524,-0.108318730037993],[0,0,0,0],[9E+09,9E+09,9E+09,9E+09,9E+09,9E+09]],
		[[1274.39345782,-188.627142215315,-30.3675026556215],[0.00942251539533556,-0.00102672230604247,-0.994071031047524,-0.108318730037993],[0,0,0,0],[9E+09,9E+09,9E+09,9E+09,9E+09,9E+09]],
		[[1274.39345782,-188.627142215315,-30.3675026556215],[0.00942251539533556,-0.00102672230604247,-0.994071031047524,-0.108318730037993],[0,0,0,0],[9E+09,9E+09,9E+09,9E+09,9E+09,9E+09]],
		[[1273.80573761255,-181.789069407022,-61.3668227324593],[0.00942251539533556,-0.00102672230604247,-0.994071031047524,-0.108318730037993],[0,0,0,0],[9E+09,9E+09,9E+09,9E+09,9E+09,9E+09]],
		[[1273.80573761255,-181.789069407022,-61.3668227324593],[0.00942251539533556,-0.00102672230604247,-0.994071031047524,-0.108318730037993],[0,0,0,0],[9E+09,9E+09,9E+09,9E+09,9E+09,9E+09]],
		[[1274.39345782,-188.627142215315,-30.3675026556215],[0.00942251539533556,-0.00102672230604247,-0.994071031047524,-0.108318730037993],[0,0,0,0],[9E+09,9E+09,9E+09,9E+09,9E+09,9E+09]],
		[[1275.33381015192,-199.568058708582,19.231409467319],[0.00942251539533556,-0.00102672230604247,-0.994071031047524,-0.108318730037993],[0,0,0,0],[9E+09,9E+09,9E+09,9E+09,9E+09,9E+09]]
		];

	!Speeds
	CONST speeddata WorkingstepSpeeddatas{140} := [
		[ 800, 500, 5000, 1000],
		[ 800, 500, 5000, 1000],
		[ 4.23333333333333, 500, 5000, 1000],
		[ 4.23333333333333, 500, 5000, 1000],
		[ 800, 500, 5000, 1000],
		[ 800, 500, 5000, 1000],
		[ 800, 500, 5000, 1000],
		[ 800, 500, 5000, 1000],
		[ 800, 500, 5000, 1000],
		[ 4.23333333333333, 500, 5000, 1000],
		[ 4.23333333333333, 500, 5000, 1000],
		[ 800, 500, 5000, 1000],
		[ 800, 500, 5000, 1000],
		[ 800, 500, 5000, 1000],
		[ 800, 500, 5000, 1000],
		[ 800, 500, 5000, 1000],
		[ 4.23333333333333, 500, 5000, 1000],
		[ 4.23333333333333, 500, 5000, 1000],
		[ 800, 500, 5000, 1000],
		[ 800, 500, 5000, 1000],
		[ 800, 500, 5000, 1000],
		[ 800, 500, 5000, 1000],
		[ 800, 500, 5000, 1000],
		[ 4.23333333333333, 500, 5000, 1000],
		[ 4.23333333333333, 500, 5000, 1000],
		[ 800, 500, 5000, 1000],
		[ 800, 500, 5000, 1000],
		[ 800, 500, 5000, 1000],
		[ 800, 500, 5000, 1000],
		[ 800, 500, 5000, 1000],
		[ 4.23333333333333, 500, 5000, 1000],
		[ 4.23333333333333, 500, 5000, 1000],
		[ 800, 500, 5000, 1000],
		[ 800, 500, 5000, 1000],
		[ 800, 500, 5000, 1000],
		[ 800, 500, 5000, 1000],
		[ 800, 500, 5000, 1000],
		[ 4.23333333333333, 500, 5000, 1000],
		[ 4.23333333333333, 500, 5000, 1000],
		[ 800, 500, 5000, 1000],
		[ 800, 500, 5000, 1000],
		[ 800, 500, 5000, 1000],
		[ 800, 500, 5000, 1000],
		[ 800, 500, 5000, 1000],
		[ 4.23333333333333, 500, 5000, 1000],
		[ 4.23333333333333, 500, 5000, 1000],
		[ 800, 500, 5000, 1000],
		[ 800, 500, 5000, 1000],
		[ 800, 500, 5000, 1000],
		[ 800, 500, 5000, 1000],
		[ 800, 500, 5000, 1000],
		[ 4.23333333333333, 500, 5000, 1000],
		[ 4.23333333333333, 500, 5000, 1000],
		[ 800, 500, 5000, 1000],
		[ 800, 500, 5000, 1000],
		[ 800, 500, 5000, 1000],
		[ 800, 500, 5000, 1000],
		[ 800, 500, 5000, 1000],
		[ 4.23333333333333, 500, 5000, 1000],
		[ 4.23333333333333, 500, 5000, 1000],
		[ 800, 500, 5000, 1000],
		[ 800, 500, 5000, 1000],
		[ 800, 500, 5000, 1000],
		[ 800, 500, 5000, 1000],
		[ 800, 500, 5000, 1000],
		[ 4.23333333333333, 500, 5000, 1000],
		[ 4.23333333333333, 500, 5000, 1000],
		[ 800, 500, 5000, 1000],
		[ 800, 500, 5000, 1000],
		[ 800, 500, 5000, 1000],
		[ 800, 500, 5000, 1000],
		[ 800, 500, 5000, 1000],
		[ 4.23333333333333, 500, 5000, 1000],
		[ 4.23333333333333, 500, 5000, 1000],
		[ 800, 500, 5000, 1000],
		[ 800, 500, 5000, 1000],
		[ 800, 500, 5000, 1000],
		[ 800, 500, 5000, 1000],
		[ 800, 500, 5000, 1000],
		[ 4.23333333333333, 500, 5000, 1000],
		[ 4.23333333333333, 500, 5000, 1000],
		[ 800, 500, 5000, 1000],
		[ 800, 500, 5000, 1000],
		[ 800, 500, 5000, 1000],
		[ 800, 500, 5000, 1000],
		[ 800, 500, 5000, 1000],
		[ 4.23333333333333, 500, 5000, 1000],
		[ 4.23333333333333, 500, 5000, 1000],
		[ 800, 500, 5000, 1000],
		[ 800, 500, 5000, 1000],
		[ 800, 500, 5000, 1000],
		[ 800, 500, 5000, 1000],
		[ 800, 500, 5000, 1000],
		[ 4.23333333333333, 500, 5000, 1000],
		[ 4.23333333333333, 500, 5000, 1000],
		[ 800, 500, 5000, 1000],
		[ 800, 500, 5000, 1000],
		[ 800, 500, 5000, 1000],
		[ 800, 500, 5000, 1000],
		[ 800, 500, 5000, 1000],
		[ 4.23333333333333, 500, 5000, 1000],
		[ 4.23333333333333, 500, 5000, 1000],
		[ 800, 500, 5000, 1000],
		[ 800, 500, 5000, 1000],
		[ 800, 500, 5000, 1000],
		[ 800, 500, 5000, 1000],
		[ 800, 500, 5000, 1000],
		[ 4.23333333333333, 500, 5000, 1000],
		[ 4.23333333333333, 500, 5000, 1000],
		[ 800, 500, 5000, 1000],
		[ 800, 500, 5000, 1000],
		[ 800, 500, 5000, 1000],
		[ 800, 500, 5000, 1000],
		[ 800, 500, 5000, 1000],
		[ 4.23333333333333, 500, 5000, 1000],
		[ 4.23333333333333, 500, 5000, 1000],
		[ 800, 500, 5000, 1000],
		[ 800, 500, 5000, 1000],
		[ 800, 500, 5000, 1000],
		[ 800, 500, 5000, 1000],
		[ 800, 500, 5000, 1000],
		[ 4.23333333333333, 500, 5000, 1000],
		[ 4.23333333333333, 500, 5000, 1000],
		[ 800, 500, 5000, 1000],
		[ 800, 500, 5000, 1000],
		[ 800, 500, 5000, 1000],
		[ 800, 500, 5000, 1000],
		[ 800, 500, 5000, 1000],
		[ 4.23333333333333, 500, 5000, 1000],
		[ 4.23333333333333, 500, 5000, 1000],
		[ 800, 500, 5000, 1000],
		[ 800, 500, 5000, 1000],
		[ 800, 500, 5000, 1000],
		[ 800, 500, 5000, 1000],
		[ 800, 500, 5000, 1000],
		[ 4.23333333333333, 500, 5000, 1000],
		[ 4.23333333333333, 500, 5000, 1000],
		[ 800, 500, 5000, 1000],
		[ 800, 500, 5000, 1000],
		[ 800, 500, 5000, 1000]
		];


ENDMODULE

--- Backups/Rob3/RAPID/TASK1/PROGMOD/CartmanWorkingPlan.mod ---
MODULE CartmanWorkingPlan
     PERS string workingPlanUUID:="sdvonvskvnwovewn342532nkfloencvosnvqwef12";
    PERS string AP238_WORKINGSTEP_NAME := "";
    PERS string AP238_WORKINGSTEP_UUID := "";
    PERS string AP238_FEATURE_NAME := "";
    PERS string AP238_FEATURE_UUID := "";
    PERS bool ok;
    PERS num startIndex :=134;
    PERS num stopIndex :=140;
      CONST speeddata serge := [ 800, 500, 5000, 1000];



    PROC main()

       !  SetDO IsDone,0;
         MoveAbsJ jHome,v400,z10,PendEff_point\WObj:=A;
        MoveAbsJ jee,v400,z10,PendEff_point\WObj:=A;
        ConfJ\Off;
        ConfL\Off;

       FOR i FROM 1 TO dim(WorkPlan,1) DO

           ok := StrToVal(Workplan{i,1}, startIndex);
           ok := StrToVal(Workplan{i,2}, stopIndex);

                WorkingStep startIndex, stopIndex, Workplan{i,3}, Workplan{i,4}, Workplan{i,5}, Workplan{i,6}, WorkingstepRobtargets, WorkingstepSpeeddatas;

        ENDFOR

        MoveAbsJ jee,v400,z10,PendEff_point\WObj:=A;
        MoveAbsJ jHome,v400,z10,PendEff_point\WObj:=A;
        !SetDO IsDone,0;
    ENDPROC

    PROC WorkingStep(num startpos, num endpos, string workingstepName, string workingstepUUID, string featureName, string featureUUID, robtarget targetList{*}, speeddata speedList{*})

        FOR i FROM startpos TO endpos DO
      !           SetDO IsDone,0;
            AP238_WORKINGSTEP_NAME := workingstepName;
            AP238_WORKINGSTEP_UUID := workingstepUUID;
            AP238_FEATURE_NAME := featureName;
            AP238_FEATURE_UUID := featureUUID;
     !       MoveL targetList{i},v1000,z100,PendEff_point\WObj:=A;
            MoveL Workingsteprobtargets{i}, speedList{i}, z100,PendEff_point\WObj:=A;
     !       SetDO IsDone,1;
            AP238_WORKINGSTEP_NAME := "";
            AP238_WORKINGSTEP_UUID := "";
            AP238_FEATURE_NAME := "";
            AP238_FEATURE_UUID := "";
        ENDFOR

    ENDPROC

ENDMODULE

--- Backups/Rob3/RAPID/TASK1/SYSMOD/WorkObjs.sys ---
MODULE WorkObjs(SYSMODULE)
    TASK PERS wobjdata A:=[FALSE,TRUE,"",[[-982.614,596.5,290.101],[1,0,0,0]],[[0,0,0],[1,0,0,0]]];
ENDMODULE

--- Backups/Rob4/RAPID/TASK1/PROGMOD/KennyTargets.mod ---
MODULE KennyTargets

	!Workplan Variables
	CONST string workplanName := "Kenny";
	CONST string workplanUUID := "4c150834-5da1-4e47-96b7-b16cde8d196c";

	!Workingsteps
	CONST string WorkPlan{20,6} := [
		["1","7", "Drilling.88", "5dba9a8c-05db-4595-a3ca-a7c776a922ef", "Hole.167", "f696efdc-798d-4b52-8da7-1cda0560be94"],
		["8","14", "Drilling.71", "36050cd1-dc9e-4879-8aed-1be84ca47fcc", "Hole.160", "7d9ff765-76db-4167-bb4c-53e49b398220"],
		["15","21", "Drilling.70", "4e2f8e6d-fe62-4a04-8e26-7213540deac3", "Hole.159", "eae91509-0626-466f-8bd8-d981c0f5cb83"],
		["22","28", "Drilling.87", "0659fa42-8109-4895-98a9-1d7bad19a7f8", "Hole.166", "d3306ec8-e7c0-4e48-ab13-ea87fff8c7f5"],
		["29","35", "Drilling.89", "25529f8b-f8c0-4dfe-8d3c-3ee9bb5aaf0b", "Hole.168", "45429ce3-7377-4a4c-ba7a-c1e998d11363"],
		["36","42", "Drilling.72", "0859f91d-f6a2-437f-b292-347030659a13", "Hole.161", "cfed41ef-af78-4deb-868f-e06b5c3e032d"],
		["43","49", "Drilling.87A", "bd213c16-608a-48e8-ba92-16dd103f0e82", "Hole.165", "e244bb89-273f-46de-9470-629b355579d0"],
		["50","56", "Drilling.72A", "30283c33-9bc4-4cb4-8bda-9191e9e1c1a8", "Hole.162", "6466e924-cde5-4cb9-be63-7b2e8a7ccfc9"],
		["57","63", "Drilling.51", "785224d9-9790-4c1a-a5a3-7fdee127c194", "Hole.149", "6ba27eaa-9f1f-4192-92ff-444f81e24c86"],
		["64","70", "Drilling.52", "6f0206cd-ac22-4230-a925-bd17b2c89fdf", "Hole.150", "7cbcafea-7ebf-4eb1-80bd-d38dc37e2ffa"],
		["71","77", "Drilling.52", "8223e776-d7de-4e22-b8f0-fb95f3561672", "Hole.151", "4113edcf-3075-48ef-82ea-78a646f36958"],
		["78","84", "Drilling.53", "15048da7-3430-4dce-a3f8-5c07c276276c", "Hole.152", "8d763157-3777-4192-8350-24f7dbecc6a9"],
		["85","91", "Drilling.66", "95c1f94a-95c9-4216-a369-009bc624fa7c", "Hole.155", "7352fd5f-6f0d-4d28-bb2c-b9767f2ea8ca"],
		["92","98", "Drilling.67", "f632f581-ae96-402c-b4f7-e3bd5086856f", "Hole.156", "7c20ef06-77fc-43ec-8049-9df34a187736"],
		["99","105", "Drilling.68", "c8ae3b54-663b-4d09-baf6-4b0ee80be638", "Hole.157", "0e7d8ffe-7fd5-4dd5-9f70-b0b78f8877dc"],
		["106","112", "Drilling.69", "d220337c-e0a3-4693-a211-54c62b6cd64b", "Hole.158", "6fcc203b-750e-4cab-906d-26d0a8242386"],
		["113","119", "Drilling.90", "f0f7cb38-96f5-48d3-840e-edf378bb551b", "Hole.170", "636bd456-6d68-43b2-b22b-21d689faa8d2"],
		["120","126", "Drilling.91", "abcac725-976e-4a50-a32b-3dd65c42f522", "Hole.171", "d8ca9eb0-5b5f-4eba-8f6d-b2fe1a9acaf1"],
		["127","133", "Drilling.92", "0d36731a-94ab-4213-8ec9-dfebb0effafd", "Hole.172", "f87e6c87-82b4-4795-8769-a91132110e61"],
		["134","140", "Drilling.93", "7777f709-fc7f-49f0-a947-dc19bdc87d5a", "Hole.173", "76d0f419-d37b-4108-8258-5a43c85176e2"]
		];

	!Positions
	CONST robtarget WorkingstepRobtargets{140} := [
		[[1251.36031479439,159.986015149395,27.4616252468863],[0.00827389312568621,0.000714793553765205,-0.996254662433507,0.0860678763663786],[0,0,0,0],[9E+09,9E+09,9E+09,9E+09,9E+09,9E+09]],
		[[1250.52908619628,151.273669125687,-22.5787992695068],[0.00827389312568621,0.000714793553765205,-0.996254662433507,0.0860678763663786],[0,0,0,0],[9E+09,9E+09,9E+09,9E+09,9E+09,9E+09]],
		[[1250.52908619628,151.273669125687,-22.5787992695068],[0.00827389312568621,0.000714793553765205,-0.996254662433507,0.0860678763663786],[0,0,0,0],[9E+09,9E+09,9E+09,9E+09,9E+09,9E+09]],
		[[1250.00956832245,145.828452860869,-53.8540645922525],[0.00827389312568621,0.000714793553765205,-0.996254662433507,0.0860678763663786],[0,0,0,0],[9E+09,9E+09,9E+09,9E+09,9E+09,9E+09]],
		[[1250.00956832245,145.828452860869,-53.8540645922525],[0.00827389312568621,0.000714793553765205,-0.996254662433507,0.0860678763663786],[0,0,0,0],[9E+09,9E+09,9E+09,9E+09,9E+09,9E+09]],
		[[1250.52908619628,151.273669125687,-22.5787992695068],[0.00827389312568621,0.000714793553765205,-0.996254662433507,0.0860678763663786],[0,0,0,0],[9E+09,9E+09,9E+09,9E+09,9E+09,9E+09]],
		[[1251.36031479439,159.986015149395,27.4616252468863],[0.00827389312568621,0.000714793553765205,-0.996254662433507,0.0860678763663786],[0,0,0,0],[9E+09,9E+09,9E+09,9E+09,9E+09,9E+09]],
		[[1190.56655432575,165.147556673713,27.5696380197376],[0.00833481880816476,0.000730999019406425,-0.996141160359995,0.0873658118059379],[0,0,0,0],[9E+09,9E+09,9E+09,9E+09,9E+09,9E+09]],
		[[1189.72949308332,156.304823646231,-22.4478129457116],[0.00833481880816476,0.000730999019406425,-0.996141160359995,0.0873658118059379],[0,0,0,0],[9E+09,9E+09,9E+09,9E+09,9E+09,9E+09]],
		[[1189.72949308332,156.304823646231,-22.4478129457116],[0.00833481880816476,0.000730999019406425,-0.996141160359995,0.0873658118059379],[0,0,0,0],[9E+09,9E+09,9E+09,9E+09,9E+09,9E+09]],
		[[1189.2063298068,150.778115504055,-53.7087197991172],[0.00833481880816476,0.000730999019406425,-0.996141160359995,0.0873658118059379],[0,0,0,0],[9E+09,9E+09,9E+09,9E+09,9E+09,9E+09]],
		[[1189.2063298068,150.778115504055,-53.7087197991172],[0.00833481880816476,0.000730999019406425,-0.996141160359995,0.0873658118059379],[0,0,0,0],[9E+09,9E+09,9E+09,9E+09,9E+09,9E+09]],
		[[1189.72949308332,156.304823646231,-22.4478129457116],[0.00833481880816476,0.000730999019406425,-0.996141160359995,0.0873658118059379],[0,0,0,0],[9E+09,9E+09,9E+09,9E+09,9E+09,9E+09]],
		[[1190.56655432575,165.147556673713,27.5696380197376],[0.00833481880816476,0.000730999019406425,-0.996141160359995,0.0873658118059379],[0,0,0,0],[9E+09,9E+09,9E+09,9E+09,9E+09,9E+09]],
		[[1191.89415560584,213.973804453541,17.5823830985576],[0.00973585929847244,0.00111256490306083,-0.993486175232847,0.113530589993472],[0,0,0,0],[9E+09,9E+09,9E+09,9E+09,9E+09,9E+09]],
		[[1190.92426864878,202.513131068111,-31.8984443484752],[0.00973585929847244,0.00111256490306083,-0.993486175232847,0.113530589993472],[0,0,0,0],[9E+09,9E+09,9E+09,9E+09,9E+09,9E+09]],
		[[1190.92426864878,202.513131068111,-31.8984443484752],[0.00973585929847244,0.00111256490306083,-0.993486175232847,0.113530589993472],[0,0,0,0],[9E+09,9E+09,9E+09,9E+09,9E+09,9E+09]],
		[[1190.31808930061,195.350210202218,-62.8239615028704],[0.00973585929847244,0.00111256490306083,-0.993486175232847,0.113530589993472],[0,0,0,0],[9E+09,9E+09,9E+09,9E+09,9E+09,9E+09]],
		[[1190.31808930061,195.350210202218,-62.8239615028704],[0.00973585929847244,0.00111256490306083,-0.993486175232847,0.113530589993472],[0,0,0,0],[9E+09,9E+09,9E+09,9E+09,9E+09,9E+09]],
		[[1190.92426864878,202.513131068111,-31.8984443484752],[0.00973585929847244,0.00111256490306083,-0.993486175232847,0.113530589993472],[0,0,0,0],[9E+09,9E+09,9E+09,9E+09,9E+09,9E+09]],
		[[1191.89415560584,213.973804453541,17.5823830985576],[0.00973585929847244,0.00111256490306083,-0.993486175232847,0.113530589993472],[0,0,0,0],[9E+09,9E+09,9E+09,9E+09,9E+09,9E+09]],
		[[1251.50868656169,112.759337427171,34.4420178830909],[0.00729205985071979,0.000442363584144468,-0.998138382466358,0.0605508020180991],[0,0,0,0],[9E+09,9E+09,9E+09,9E+09,9E+09,9E+09]],
		[[1250.77191390728,106.618500806138,-15.9800734226999],[0.00729205985071979,0.000442363584144468,-0.998138382466358,0.0605508020180991],[0,0,0,0],[9E+09,9E+09,9E+09,9E+09,9E+09,9E+09]],
		[[1250.77191390728,106.618500806138,-15.9800734226999],[0.00729205985071979,0.000442363584144468,-0.998138382466358,0.0605508020180991],[0,0,0,0],[9E+09,9E+09,9E+09,9E+09,9E+09,9E+09]],
		[[1250.31143099827,102.780477917993,-47.4938804888192],[0.00729205985071979,0.000442363584144468,-0.998138382466358,0.0605508020180991],[0,0,0,0],[9E+09,9E+09,9E+09,9E+09,9E+09,9E+09]],
		[[1250.31143099827,102.780477917993,-47.4938804888192],[0.00729205985071979,0.000442363584144468,-0.998138382466358,0.0605508020180991],[0,0,0,0],[9E+09,9E+09,9E+09,9E+09,9E+09,9E+09]],
		[[1250.77191390728,106.618500806138,-15.9800734226999],[0.00729205985071979,0.000442363584144468,-0.998138382466358,0.0605508020180991],[0,0,0,0],[9E+09,9E+09,9E+09,9E+09,9E+09,9E+09]],
		[[1251.50868656169,112.759337427171,34.4420178830909],[0.00729205985071979,0.000442363584144468,-0.998138382466358,0.0605508020180991],[0,0,0,0],[9E+09,9E+09,9E+09,9E+09,9E+09,9E+09]],
		[[1251.8601825108,210.524561887497,17.2060251950538],[0.0097362625680173,0.00111307904909481,-0.993480782143631,0.113577734426767],[0,0,0,0],[9E+09,9E+09,9E+09,9E+09,9E+09,9E+09]],
		[[1250.89027144533,199.059191507408,-32.2737136338089],[0.0097362625680173,0.00111307904909481,-0.993480782143631,0.113577734426767],[0,0,0,0],[9E+09,9E+09,9E+09,9E+09,9E+09,9E+09]],
		[[1250.89027144533,199.059191507408,-32.2737136338089],[0.0097362625680173,0.00111307904909481,-0.993480782143631,0.113577734426767],[0,0,0,0],[9E+09,9E+09,9E+09,9E+09,9E+09,9E+09]],
		[[1250.28407702942,191.893335019853,-63.1985504018481],[0.0097362625680173,0.00111307904909481,-0.993480782143631,0.113577734426767],[0,0,0,0],[9E+09,9E+09,9E+09,9E+09,9E+09,9E+09]],
		[[1250.28407702942,191.893335019853,-63.1985504018481],[0.0097362625680173,0.00111307904909481,-0.993480782143631,0.113577734426767],[0,0,0,0],[9E+09,9E+09,9E+09,9E+09,9E+09,9E+09]],
		[[1250.89027144533,199.059191507408,-32.2737136338089],[0.0097362625680173,0.00111307904909481,-0.993480782143631,0.113577734426767],[0,0,0,0],[9E+09,9E+09,9E+09,9E+09,9E+09,9E+09]],
		[[1251.8601825108,210.524561887497,17.2060251950538],[0.0097362625680173,0.00111307904909481,-0.993480782143631,0.113577734426767],[0,0,0,0],[9E+09,9E+09,9E+09,9E+09,9E+09,9E+09]],
		[[1190.88023867958,116.257500079554,34.9005826267419],[0.00731948636979851,0.000450203628618277,-0.998086922900926,0.0613898751435108],[0,0,0,0],[9E+09,9E+09,9E+09,9E+09,9E+09,9E+09]],
		[[1190.14080955814,110.031886232754,-15.5110725415314],[0.00731948636979851,0.000450203628618277,-0.998086922900926,0.0613898751435108],[0,0,0,0],[9E+09,9E+09,9E+09,9E+09,9E+09,9E+09]],
		[[1190.14080955814,110.031886232754,-15.5110725415314],[0.00731948636979851,0.000450203628618277,-0.998086922900926,0.0613898751435108],[0,0,0,0],[9E+09,9E+09,9E+09,9E+09,9E+09,9E+09]],
		[[1189.67866635724,106.140877578504,-47.0183570217021],[0.00731948636979851,0.000450203628618277,-0.998086922900926,0.0613898751435108],[0,0,0,0],[9E+09,9E+09,9E+09,9E+09,9E+09,9E+09]],
		[[1189.67866635724,106.140877578504,-47.0183570217021],[0.00731948636979851,0.000450203628618277,-0.998086922900926,0.0613898751435108],[0,0,0,0],[9E+09,9E+09,9E+09,9E+09,9E+09,9E+09]],
		[[1190.14080955814,110.031886232754,-15.5110725415314],[0.00731948636979851,0.000450203628618277,-0.998086922900926,0.0613898751435108],[0,0,0,0],[9E+09,9E+09,9E+09,9E+09,9E+09,9E+09]],
		[[1190.88023867958,116.257500079554,34.9005826267419],[0.00731948636979851,0.000450203628618277,-0.998086922900926,0.0613898751435108],[0,0,0,0],[9E+09,9E+09,9E+09,9E+09,9E+09,9E+09]],
		[[1250.76447640153,68.6402546108708,38.7643104755585],[0.00669120018047459,0.000246507461145111,-0.999299675598547,0.0368147446392719],[0,0,0,0],[9E+09,9E+09,9E+09,9E+09,9E+09,9E+09]],
		[[1250.08604859299,64.9023284513774,-11.8934396100383],[0.00669120018047459,0.000246507461145111,-0.999299675598547,0.0368147446392719],[0,0,0,0],[9E+09,9E+09,9E+09,9E+09,9E+09,9E+09]],
		[[1250.08604859299,64.9023284513774,-11.8934396100383],[0.00669120018047459,0.000246507461145111,-0.999299675598547,0.0368147446392719],[0,0,0,0],[9E+09,9E+09,9E+09,9E+09,9E+09,9E+09]],
		[[1249.66203121265,62.5661246016938,-43.5545334135362],[0.00669120018047459,0.000246507461145111,-0.999299675598547,0.0368147446392719],[0,0,0,0],[9E+09,9E+09,9E+09,9E+09,9E+09,9E+09]],
		[[1249.66203121265,62.5661246016938,-43.5545334135362],[0.00669120018047459,0.000246507461145111,-0.999299675598547,0.0368147446392719],[0,0,0,0],[9E+09,9E+09,9E+09,9E+09,9E+09,9E+09]],
		[[1250.08604859299,64.9023284513774,-11.8934396100383],[0.00669120018047459,0.000246507461145111,-0.999299675598547,0.0368147446392719],[0,0,0,0],[9E+09,9E+09,9E+09,9E+09,9E+09,9E+09]],
		[[1250.76447640153,68.6402546108708,38.7643104755585],[0.00669120018047459,0.000246507461145111,-0.999299675598547,0.0368147446392719],[0,0,0,0],[9E+09,9E+09,9E+09,9E+09,9E+09,9E+09]],
		[[1189.9772715838,69.4582698852428,39.5179868929106],[0.00668793620390687,0.000245146305514718,-0.999306502156587,0.0366295803987568],[0,0,0,0],[9E+09,9E+09,9E+09,9E+09,9E+09,9E+09]],
		[[1189.29916082133,65.7391188387643,-11.1411493145624],[0.00668793620390687,0.000245146305514718,-0.999306502156587,0.0366295803987568],[0,0,0,0],[9E+09,9E+09,9E+09,9E+09,9E+09,9E+09]],
		[[1189.29916082133,65.7391188387643,-11.1411493145624],[0.00668793620390687,0.000245146305514718,-0.999306502156587,0.0366295803987568],[0,0,0,0],[9E+09,9E+09,9E+09,9E+09,9E+09,9E+09]],
		[[1188.87534159478,63.4146494347152,-42.803109444233],[0.00668793620390687,0.000245146305514718,-0.999306502156587,0.0366295803987568],[0,0,0,0],[9E+09,9E+09,9E+09,9E+09,9E+09,9E+09]],
		[[1188.87534159478,63.4146494347152,-42.803109444233],[0.00668793620390687,0.000245146305514718,-0.999306502156587,0.0366295803987568],[0,0,0,0],[9E+09,9E+09,9E+09,9E+09,9E+09,9E+09]],
		[[1189.29916082133,65.7391188387643,-11.1411493145624],[0.00668793620390687,0.000245146305514718,-0.999306502156587,0.0366295803987568],[0,0,0,0],[9E+09,9E+09,9E+09,9E+09,9E+09,9E+09]],
		[[1189.9772715838,69.4582698852428,39.5179868929106],[0.00668793620390687,0.000245146305514718,-0.999306502156587,0.0366295803987568],[0,0,0,0],[9E+09,9E+09,9E+09,9E+09,9E+09,9E+09]],
		[[1048.75377702369,221.064248736861,18.7456359573398],[0.00969862451718228,0.0011013674490227,-0.993566525165611,0.112828559073272],[0,0,0,0],[9E+09,9E+09,9E+09,9E+09,9E+09,9E+09]],
		[[1047.78736158715,209.673531246336,-30.7514103813565],[0.00969862451718228,0.0011013674490227,-0.993566525165611,0.112828559073272],[0,0,0,0],[9E+09,9E+09,9E+09,9E+09,9E+09,9E+09]],
		[[1047.78736158715,209.673531246336,-30.7514103813565],[0.00969862451718228,0.0011013674490227,-0.993566525165611,0.112828559073272],[0,0,0,0],[9E+09,9E+09,9E+09,9E+09,9E+09,9E+09]],
		[[1047.18335193931,202.554332814758,-61.6870643430416],[0.00969862451718228,0.0011013674490227,-0.993566525165611,0.112828559073272],[0,0,0,0],[9E+09,9E+09,9E+09,9E+09,9E+09,9E+09]],
		[[1047.18335193931,202.554332814758,-61.6870643430416],[0.00969862451718228,0.0011013674490227,-0.993566525165611,0.112828559073272],[0,0,0,0],[9E+09,9E+09,9E+09,9E+09,9E+09,9E+09]],
		[[1047.78736158715,209.673531246336,-30.7514103813565],[0.00969862451718228,0.0011013674490227,-0.993566525165611,0.112828559073272],[0,0,0,0],[9E+09,9E+09,9E+09,9E+09,9E+09,9E+09]],
		[[1048.75377702369,221.064248736861,18.7456359573398],[0.00969862451718228,0.0011013674490227,-0.993566525165611,0.112828559073272],[0,0,0,0],[9E+09,9E+09,9E+09,9E+09,9E+09,9E+09]],
		[[1049.72266482233,161.388258470636,30.5369306758237],[0.00810433453815839,0.000668070226723706,-0.996586609691307,0.0821523148051996],[0,0,0,0],[9E+09,9E+09,9E+09,9E+09,9E+09,9E+09]],
		[[1048.90765118534,153.069523657326,-19.5706975246546],[0.00810433453815839,0.000668070226723706,-0.996586609691307,0.0821523148051996],[0,0,0,0],[9E+09,9E+09,9E+09,9E+09,9E+09,9E+09]],
		[[1048.90765118534,153.069523657326,-19.5706975246546],[0.00810433453815839,0.000668070226723706,-0.996586609691307,0.0821523148051996],[0,0,0,0],[9E+09,9E+09,9E+09,9E+09,9E+09,9E+09]],
		[[1048.39826766222,147.870314399008,-50.8879651499535],[0.00810433453815839,0.000668070226723706,-0.996586609691307,0.0821523148051996],[0,0,0,0],[9E+09,9E+09,9E+09,9E+09,9E+09,9E+09]],
		[[1048.39826766222,147.870314399008,-50.8879651499535],[0.00810433453815839,0.000668070226723706,-0.996586609691307,0.0821523148051996],[0,0,0,0],[9E+09,9E+09,9E+09,9E+09,9E+09,9E+09]],
		[[1048.90765118534,153.069523657326,-19.5706975246546],[0.00810433453815839,0.000668070226723706,-0.996586609691307,0.0821523148051996],[0,0,0,0],[9E+09,9E+09,9E+09,9E+09,9E+09,9E+09]],
		[[1049.72266482233,161.388258470636,30.5369306758237],[0.00810433453815839,0.000668070226723706,-0.996586609691307,0.0821523148051996],[0,0,0,0],[9E+09,9E+09,9E+09,9E+09,9E+09,9E+09]],
		[[1050.01208432635,107.933890240474,37.9095374224083],[0.007122245347503,0.00039121136422263,-0.998469455496607,0.0548440244255241],[0,0,0,0],[9E+09,9E+09,9E+09,9E+09,9E+09,9E+09]],
		[[1049.29175162139,102.369982698389,-12.5797094887637],[0.007122245347503,0.00039121136422263,-0.998469455496607,0.0548440244255241],[0,0,0,0],[9E+09,9E+09,9E+09,9E+09,9E+09,9E+09]],
		[[1049.29175162139,102.369982698389,-12.5797094887637],[0.007122245347503,0.00039121136422263,-0.998469455496607,0.0548440244255241],[0,0,0,0],[9E+09,9E+09,9E+09,9E+09,9E+09,9E+09]],
		[[1048.84154368078,98.8925404845857,-44.1354888082459],[0.007122245347503,0.00039121136422263,-0.998469455496607,0.0548440244255241],[0,0,0,0],[9E+09,9E+09,9E+09,9E+09,9E+09,9E+09]],
		[[1048.84154368078,98.8925404845857,-44.1354888082459],[0.007122245347503,0.00039121136422263,-0.998469455496607,0.0548440244255241],[0,0,0,0],[9E+09,9E+09,9E+09,9E+09,9E+09,9E+09]],
		[[1049.29175162139,102.369982698389,-12.5797094887637],[0.007122245347503,0.00039121136422263,-0.998469455496607,0.0548440244255241],[0,0,0,0],[9E+09,9E+09,9E+09,9E+09,9E+09,9E+09]],
		[[1050.01208432635,107.933890240474,37.9095374224083],[0.007122245347503,0.00039121136422263,-0.998469455496607,0.0548440244255241],[0,0,0,0],[9E+09,9E+09,9E+09,9E+09,9E+09,9E+09]],
		[[1048.45280482734,61.188425000286,41.9579660547863],[0.00659046299640987,0.00020471594525679,-0.999496183042603,0.0310468029294715],[0,0,0,0],[9E+09,9E+09,9E+09,9E+09,9E+09,9E+09]],
		[[1047.78419688503,58.0355219643173,-8.73968838666952],[0.00659046299640987,0.00020471594525679,-0.999496183042603,0.0310468029294715],[0,0,0,0],[9E+09,9E+09,9E+09,9E+09,9E+09,9E+09]],
		[[1047.78419688503,58.0355219643173,-8.73968838666952],[0.00659046299640987,0.00020471594525679,-0.999496183042603,0.0310468029294715],[0,0,0,0],[9E+09,9E+09,9E+09,9E+09,9E+09,9E+09]],
		[[1047.36631692108,56.064957566837,-40.4257224125791],[0.00659046299640987,0.00020471594525679,-0.999496183042603,0.0310468029294715],[0,0,0,0],[9E+09,9E+09,9E+09,9E+09,9E+09,9E+09]],
		[[1047.36631692108,56.064957566837,-40.4257224125791],[0.00659046299640987,0.00020471594525679,-0.999496183042603,0.0310468029294715],[0,0,0,0],[9E+09,9E+09,9E+09,9E+09,9E+09,9E+09]],
		[[1047.78419688503,58.0355219643173,-8.73968838666952],[0.00659046299640987,0.00020471594525679,-0.999496183042603,0.0310468029294715],[0,0,0,0],[9E+09,9E+09,9E+09,9E+09,9E+09,9E+09]],
		[[1048.45280482734,61.188425000286,41.9579660547863],[0.00659046299640987,0.00020471594525679,-0.999496183042603,0.0310468029294715],[0,0,0,0],[9E+09,9E+09,9E+09,9E+09,9E+09,9E+09]],
		[[1124.58450857921,76.9515299774283,39.8228669588901],[0.00675250584078808,0.000269433238042634,-0.999182078945179,0.0398685864483636],[0,0,0,0],[9E+09,9E+09,9E+09,9E+09,9E+09,9E+09]],
		[[1123.90010650359,72.904009858962,-10.8110068282249],[0.00675250584078808,0.000269433238042634,-0.999182078945179,0.0398685864483636],[0,0,0,0],[9E+09,9E+09,9E+09,9E+09,9E+09,9E+09]],
		[[1123.90010650359,72.904009858962,-10.8110068282249],[0.00675250584078808,0.000269433238042634,-0.999182078945179,0.0398685864483636],[0,0,0,0],[9E+09,9E+09,9E+09,9E+09,9E+09,9E+09]],
		[[1123.47235520633,70.3743097849206,-42.457177945172],[0.00675250584078808,0.000269433238042634,-0.999182078945179,0.0398685864483636],[0,0,0,0],[9E+09,9E+09,9E+09,9E+09,9E+09,9E+09]],
		[[1123.47235520633,70.3743097849206,-42.457177945172],[0.00675250584078808,0.000269433238042634,-0.999182078945179,0.0398685864483636],[0,0,0,0],[9E+09,9E+09,9E+09,9E+09,9E+09,9E+09]],
		[[1123.90010650359,72.904009858962,-10.8110068282249],[0.00675250584078808,0.000269433238042634,-0.999182078945179,0.0398685864483636],[0,0,0,0],[9E+09,9E+09,9E+09,9E+09,9E+09,9E+09]],
		[[1124.58450857921,76.9515299774283,39.8228669588901],[0.00675250584078808,0.000269433238042634,-0.999182078945179,0.0398685864483636],[0,0,0,0],[9E+09,9E+09,9E+09,9E+09,9E+09,9E+09]],
		[[1126.5993688537,133.371202707924,33.609656791981],[0.00758868592259089,0.000526723182265742,-0.997570999567389,0.0692404161655443],[0,0,0,0],[9E+09,9E+09,9E+09,9E+09,9E+09,9E+09]],
		[[1125.83393655486,126.353057912489,-16.6973979521224],[0.00758868592259089,0.000526723182265742,-0.997570999567389,0.0692404161655443],[0,0,0,0],[9E+09,9E+09,9E+09,9E+09,9E+09,9E+09]],
		[[1125.83393655486,126.353057912489,-16.6973979521224],[0.00758868592259089,0.000526723182265742,-0.997570999567389,0.0692404161655443],[0,0,0,0],[9E+09,9E+09,9E+09,9E+09,9E+09,9E+09]],
		[[1125.35554136809,121.966717415342,-48.139307167187],[0.00758868592259089,0.000526723182265742,-0.997570999567389,0.0692404161655443],[0,0,0,0],[9E+09,9E+09,9E+09,9E+09,9E+09,9E+09]],
		[[1125.35554136809,121.966717415342,-48.139307167187],[0.00758868592259089,0.000526723182265742,-0.997570999567389,0.0692404161655443],[0,0,0,0],[9E+09,9E+09,9E+09,9E+09,9E+09,9E+09]],
		[[1125.83393655486,126.353057912489,-16.6973979521224],[0.00758868592259089,0.000526723182265742,-0.997570999567389,0.0692404161655443],[0,0,0,0],[9E+09,9E+09,9E+09,9E+09,9E+09,9E+09]],
		[[1126.5993688537,133.371202707924,33.609656791981],[0.00758868592259089,0.000526723182265742,-0.997570999567389,0.0692404161655443],[0,0,0,0],[9E+09,9E+09,9E+09,9E+09,9E+09,9E+09]],
		[[1126.0616372464,186.211885781352,24.7464515853499],[0.00880082191675858,0.000856592596021549,-0.995257819874454,0.0968694160272657],[0,0,0,0],[9E+09,9E+09,9E+09,9E+09,9E+09,9E+09]],
		[[1125.18014455072,176.41585939664,-25.0922967706981],[0.00880082191675858,0.000856592596021549,-0.995257819874454,0.0968694160272657],[0,0,0,0],[9E+09,9E+09,9E+09,9E+09,9E+09,9E+09]],
		[[1125.18014455072,176.41585939664,-25.0922967706981],[0.00880082191675858,0.000856592596021549,-0.995257819874454,0.0968694160272657],[0,0,0,0],[9E+09,9E+09,9E+09,9E+09,9E+09,9E+09]],
		[[1124.62921161592,170.293342906194,-56.2415144932284],[0.00880082191675858,0.000856592596021549,-0.995257819874454,0.0968694160272657],[0,0,0,0],[9E+09,9E+09,9E+09,9E+09,9E+09,9E+09]],
		[[1124.62921161592,170.293342906194,-56.2415144932284],[0.00880082191675858,0.000856592596021549,-0.995257819874454,0.0968694160272657],[0,0,0,0],[9E+09,9E+09,9E+09,9E+09,9E+09,9E+09]],
		[[1125.18014455072,176.41585939664,-25.0922967706981],[0.00880082191675858,0.000856592596021549,-0.995257819874454,0.0968694160272657],[0,0,0,0],[9E+09,9E+09,9E+09,9E+09,9E+09,9E+09]],
		[[1126.0616372464,186.211885781352,24.7464515853499],[0.00880082191675858,0.000856592596021549,-0.995257819874454,0.0968694160272657],[0,0,0,0],[9E+09,9E+09,9E+09,9E+09,9E+09,9E+09]],
		[[1124.84625477698,220.957336979353,17.2741397681532],[0.0098367962378513,0.00114012296637116,-0.993301363012953,0.115127493658146],[0,0,0,0],[9E+09,9E+09,9E+09,9E+09,9E+09,9E+09]],
		[[1123.86686698609,209.337597808087,-32.1693882324538],[0.0098367962378513,0.00114012296637116,-0.993301363012953,0.115127493658146],[0,0,0,0],[9E+09,9E+09,9E+09,9E+09,9E+09,9E+09]],
		[[1123.86686698609,209.337597808087,-32.1693882324538],[0.0098367962378513,0.00114012296637116,-0.993301363012953,0.115127493658146],[0,0,0,0],[9E+09,9E+09,9E+09,9E+09,9E+09,9E+09]],
		[[1123.25474961678,202.075260826046,-63.071593232833],[0.0098367962378513,0.00114012296637116,-0.993301363012953,0.115127493658146],[0,0,0,0],[9E+09,9E+09,9E+09,9E+09,9E+09,9E+09]],
		[[1123.25474961678,202.075260826046,-63.071593232833],[0.0098367962378513,0.00114012296637116,-0.993301363012953,0.115127493658146],[0,0,0,0],[9E+09,9E+09,9E+09,9E+09,9E+09,9E+09]],
		[[1123.86686698609,209.337597808087,-32.1693882324538],[0.0098367962378513,0.00114012296637116,-0.993301363012953,0.115127493658146],[0,0,0,0],[9E+09,9E+09,9E+09,9E+09,9E+09,9E+09]],
		[[1124.84625477698,220.957336979353,17.2741397681532],[0.0098367962378513,0.00114012296637116,-0.993301363012953,0.115127493658146],[0,0,0,0],[9E+09,9E+09,9E+09,9E+09,9E+09,9E+09]],
		[[1286.40443376685,208.720093463579,16.9470304734434],[0.00974259835249316,0.00111507411475759,-0.993466087636441,0.113705633560541],[0,0,0,0],[9E+09,9E+09,9E+09,9E+09,9E+09,9E+09]],
		[[1285.43393523947,197.241980312679,-32.5297423710288],[0.00974259835249316,0.00111507411475759,-0.993466087636441,0.113705633560541],[0,0,0,0],[9E+09,9E+09,9E+09,9E+09,9E+09,9E+09]],
		[[1285.43393523947,197.241980312679,-32.5297423710288],[0.00974259835249316,0.00111507411475759,-0.993466087636441,0.113705633560541],[0,0,0,0],[9E+09,9E+09,9E+09,9E+09,9E+09,9E+09]],
		[[1284.82737365986,190.068159593366,-63.4527253988237],[0.00974259835249316,0.00111507411475759,-0.993466087636441,0.113705633560541],[0,0,0,0],[9E+09,9E+09,9E+09,9E+09,9E+09,9E+09]],
		[[1284.82737365986,190.068159593366,-63.4527253988237],[0.00974259835249316,0.00111507411475759,-0.993466087636441,0.113705633560541],[0,0,0,0],[9E+09,9E+09,9E+09,9E+09,9E+09,9E+09]],
		[[1285.43393523947,197.241980312679,-32.5297423710288],[0.00974259835249316,0.00111507411475759,-0.993466087636441,0.113705633560541],[0,0,0,0],[9E+09,9E+09,9E+09,9E+09,9E+09,9E+09]],
		[[1286.40443376685,208.720093463579,16.9470304734434],[0.00974259835249316,0.00111507411475759,-0.993466087636441,0.113705633560541],[0,0,0,0],[9E+09,9E+09,9E+09,9E+09,9E+09,9E+09]],
		[[1286.33124649681,153.926988279123,27.9242514810087],[0.00816312780487694,0.000684952269338226,-0.996464762410529,0.0836114313892439],[0,0,0,0],[9E+09,9E+09,9E+09,9E+09,9E+09,9E+09]],
		[[1285.51062336092,145.461530334075,-22.1587056945564],[0.00816312780487694,0.000684952269338226,-0.996464762410529,0.0836114313892439],[0,0,0,0],[9E+09,9E+09,9E+09,9E+09,9E+09,9E+09]],
		[[1285.51062336092,145.461530334075,-22.1587056945564],[0.00816312780487694,0.000684952269338226,-0.996464762410529,0.0836114313892439],[0,0,0,0],[9E+09,9E+09,9E+09,9E+09,9E+09,9E+09]],
		[[1284.997733901,140.170619118421,-53.4605539292846],[0.00816312780487694,0.000684952269338226,-0.996464762410529,0.0836114313892439],[0,0,0,0],[9E+09,9E+09,9E+09,9E+09,9E+09,9E+09]],
		[[1284.997733901,140.170619118421,-53.4605539292846],[0.00816312780487694,0.000684952269338226,-0.996464762410529,0.0836114313892439],[0,0,0,0],[9E+09,9E+09,9E+09,9E+09,9E+09,9E+09]],
		[[1285.51062336092,145.461530334075,-22.1587056945564],[0.00816312780487694,0.000684952269338226,-0.996464762410529,0.0836114313892439],[0,0,0,0],[9E+09,9E+09,9E+09,9E+09,9E+09,9E+09]],
		[[1286.33124649681,153.926988279123,27.9242514810087],[0.00816312780487694,0.000684952269338226,-0.996464762410529,0.0836114313892439],[0,0,0,0],[9E+09,9E+09,9E+09,9E+09,9E+09,9E+09]],
		[[1280.46270299124,102.38309339464,35.2332574820644],[0.00713645430881742,0.0003960721694737,-0.998437927952443,0.055413158841264],[0,0,0,0],[9E+09,9E+09,9E+09,9E+09,9E+09,9E+09]],
		[[1279.74100171248,96.7616237083952,-15.2495933272039],[0.00713645430881742,0.0003960721694737,-0.998437927952443,0.055413158841264],[0,0,0,0],[9E+09,9E+09,9E+09,9E+09,9E+09,9E+09]],
		[[1279.74100171248,96.7616237083952,-15.2495933272039],[0.00713645430881742,0.0003960721694737,-0.998437927952443,0.055413158841264],[0,0,0,0],[9E+09,9E+09,9E+09,9E+09,9E+09,9E+09]],
		[[1279.28993841325,93.2482051544925,-46.8013750829966],[0.00713645430881742,0.0003960721694737,-0.998437927952443,0.055413158841264],[0,0,0,0],[9E+09,9E+09,9E+09,9E+09,9E+09,9E+09]],
		[[1279.28993841325,93.2482051544925,-46.8013750829966],[0.00713645430881742,0.0003960721694737,-0.998437927952443,0.055413158841264],[0,0,0,0],[9E+09,9E+09,9E+09,9E+09,9E+09,9E+09]],
		[[1279.74100171248,96.7616237083952,-15.2495933272039],[0.00713645430881742,0.0003960721694737,-0.998437927952443,0.055413158841264],[0,0,0,0],[9E+09,9E+09,9E+09,9E+09,9E+09,9E+09]],
		[[1280.46270299124,102.38309339464,35.2332574820644],[0.00713645430881742,0.0003960721694737,-0.998437927952443,0.055413158841264],[0,0,0,0],[9E+09,9E+09,9E+09,9E+09,9E+09,9E+09]],
		[[1279.80555575599,62.0258838013912,38.8434555023548],[0.00663132377542586,0.000222501158844028,-0.999415571315941,0.0335334437457661],[0,0,0,0],[9E+09,9E+09,9E+09,9E+09,9E+09,9E+09]],
		[[1279.13296507583,58.6207271556254,-11.8378283211116],[0.00663132377542586,0.000222501158844028,-0.999415571315941,0.0335334437457661],[0,0,0,0],[9E+09,9E+09,9E+09,9E+09,9E+09,9E+09]],
		[[1279.13296507583,58.6207271556254,-11.8378283211116],[0.00663132377542586,0.000222501158844028,-0.999415571315941,0.0335334437457661],[0,0,0,0],[9E+09,9E+09,9E+09,9E+09,9E+09,9E+09]],
		[[1278.71259590072,56.4925042520218,-43.5136307107779],[0.00663132377542586,0.000222501158844028,-0.999415571315941,0.0335334437457661],[0,0,0,0],[9E+09,9E+09,9E+09,9E+09,9E+09,9E+09]],
		[[1278.71259590072,56.4925042520218,-43.5136307107779],[0.00663132377542586,0.000222501158844028,-0.999415571315941,0.0335334437457661],[0,0,0,0],[9E+09,9E+09,9E+09,9E+09,9E+09,9E+09]],
		[[1279.13296507583,58.6207271556254,-11.8378283211116],[0.00663132377542586,0.000222501158844028,-0.999415571315941,0.0335334437457661],[0,0,0,0],[9E+09,9E+09,9E+09,9E+09,9E+09,9E+09]],
		[[1279.80555575599,62.0258838013912,38.8434555023548],[0.00663132377542586,0.000222501158844028,-0.999415571315941,0.0335334437457661],[0,0,0,0],[9E+09,9E+09,9E+09,9E+09,9E+09,9E+09]]
		];

	!Speeds
	CONST speeddata WorkingstepSpeeddatas{140} := [
		[ 800, 500, 5000, 1000],
		[ 800, 500, 5000, 1000],
		[ 4.23333333333333, 500, 5000, 1000],
		[ 4.23333333333333, 500, 5000, 1000],
		[ 800, 500, 5000, 1000],
		[ 800, 500, 5000, 1000],
		[ 800, 500, 5000, 1000],
		[ 800, 500, 5000, 1000],
		[ 800, 500, 5000, 1000],
		[ 4.23333333333333, 500, 5000, 1000],
		[ 4.23333333333333, 500, 5000, 1000],
		[ 800, 500, 5000, 1000],
		[ 800, 500, 5000, 1000],
		[ 800, 500, 5000, 1000],
		[ 800, 500, 5000, 1000],
		[ 800, 500, 5000, 1000],
		[ 4.23333333333333, 500, 5000, 1000],
		[ 4.23333333333333, 500, 5000, 1000],
		[ 800, 500, 5000, 1000],
		[ 800, 500, 5000, 1000],
		[ 800, 500, 5000, 1000],
		[ 800, 500, 5000, 1000],
		[ 800, 500, 5000, 1000],
		[ 4.23333333333333, 500, 5000, 1000],
		[ 4.23333333333333, 500, 5000, 1000],
		[ 800, 500, 5000, 1000],
		[ 800, 500, 5000, 1000],
		[ 800, 500, 5000, 1000],
		[ 800, 500, 5000, 1000],
		[ 800, 500, 5000, 1000],
		[ 4.23333333333333, 500, 5000, 1000],
		[ 4.23333333333333, 500, 5000, 1000],
		[ 800, 500, 5000, 1000],
		[ 800, 500, 5000, 1000],
		[ 800, 500, 5000, 1000],
		[ 800, 500, 5000, 1000],
		[ 800, 500, 5000, 1000],
		[ 4.23333333333333, 500, 5000, 1000],
		[ 4.23333333333333, 500, 5000, 1000],
		[ 800, 500, 5000, 1000],
		[ 800, 500, 5000, 1000],
		[ 800, 500, 5000, 1000],
		[ 800, 500, 5000, 1000],
		[ 800, 500, 5000, 1000],
		[ 4.23333333333333, 500, 5000, 1000],
		[ 4.23333333333333, 500, 5000, 1000],
		[ 800, 500, 5000, 1000],
		[ 800, 500, 5000, 1000],
		[ 800, 500, 5000, 1000],
		[ 800, 500, 5000, 1000],
		[ 800, 500, 5000, 1000],
		[ 4.23333333333333, 500, 5000, 1000],
		[ 4.23333333333333, 500, 5000, 1000],
		[ 800, 500, 5000, 1000],
		[ 800, 500, 5000, 1000],
		[ 800, 500, 5000, 1000],
		[ 800, 500, 5000, 1000],
		[ 800, 500, 5000, 1000],
		[ 4.23333333333333, 500, 5000, 1000],
		[ 4.23333333333333, 500, 5000, 1000],
		[ 800, 500, 5000, 1000],
		[ 800, 500, 5000, 1000],
		[ 800, 500, 5000, 1000],
		[ 800, 500, 5000, 1000],
		[ 800, 500, 5000, 1000],
		[ 4.23333333333333, 500, 5000, 1000],
		[ 4.23333333333333, 500, 5000, 1000],
		[ 800, 500, 5000, 1000],
		[ 800, 500, 5000, 1000],
		[ 800, 500, 5000, 1000],
		[ 800, 500, 5000, 1000],
		[ 800, 500, 5000, 1000],
		[ 4.23333333333333, 500, 5000, 1000],
		[ 4.23333333333333, 500, 5000, 1000],
		[ 800, 500, 5000, 1000],
		[ 800, 500, 5000, 1000],
		[ 800, 500, 5000, 1000],
		[ 800, 500, 5000, 1000],
		[ 800, 500, 5000, 1000],
		[ 4.23333333333333, 500, 5000, 1000],
		[ 4.23333333333333, 500, 5000, 1000],
		[ 800, 500, 5000, 1000],
		[ 800, 500, 5000, 1000],
		[ 800, 500, 5000, 1000],
		[ 800, 500, 5000, 1000],
		[ 800, 500, 5000, 1000],
		[ 4.23333333333333, 500, 5000, 1000],
		[ 4.23333333333333, 500, 5000, 1000],
		[ 800, 500, 5000, 1000],
		[ 800, 500, 5000, 1000],
		[ 800, 500, 5000, 1000],
		[ 800, 500, 5000, 1000],
		[ 800, 500, 5000, 1000],
		[ 4.23333333333333, 500, 5000, 1000],
		[ 4.23333333333333, 500, 5000, 1000],
		[ 800, 500, 5000, 1000],
		[ 800, 500, 5000, 1000],
		[ 800, 500, 5000, 1000],
		[ 800, 500, 5000, 1000],
		[ 800, 500, 5000, 1000],
		[ 4.23333333333333, 500, 5000, 1000],
		[ 4.23333333333333, 500, 5000, 1000],
		[ 800, 500, 5000, 1000],
		[ 800, 500, 5000, 1000],
		[ 800, 500, 5000, 1000],
		[ 800, 500, 5000, 1000],
		[ 800, 500, 5000, 1000],
		[ 4.23333333333333, 500, 5000, 1000],
		[ 4.23333333333333, 500, 5000, 1000],
		[ 800, 500, 5000, 1000],
		[ 800, 500, 5000, 1000],
		[ 800, 500, 5000, 1000],
		[ 800, 500, 5000, 1000],
		[ 800, 500, 5000, 1000],
		[ 4.23333333333333, 500, 5000, 1000],
		[ 4.23333333333333, 500, 5000, 1000],
		[ 800, 500, 5000, 1000],
		[ 800, 500, 5000, 1000],
		[ 800, 500, 5000, 1000],
		[ 800, 500, 5000, 1000],
		[ 800, 500, 5000, 1000],
		[ 4.23333333333333, 500, 5000, 1000],
		[ 4.23333333333333, 500, 5000, 1000],
		[ 800, 500, 5000, 1000],
		[ 800, 500, 5000, 1000],
		[ 800, 500, 5000, 1000],
		[ 800, 500, 5000, 1000],
		[ 800, 500, 5000, 1000],
		[ 4.23333333333333, 500, 5000, 1000],
		[ 4.23333333333333, 500, 5000, 1000],
		[ 800, 500, 5000, 1000],
		[ 800, 500, 5000, 1000],
		[ 800, 500, 5000, 1000],
		[ 800, 500, 5000, 1000],
		[ 800, 500, 5000, 1000],
		[ 4.23333333333333, 500, 5000, 1000],
		[ 4.23333333333333, 500, 5000, 1000],
		[ 800, 500, 5000, 1000],
		[ 800, 500, 5000, 1000],
		[ 800, 500, 5000, 1000]
		];


ENDMODULE

--- Backups/Rob4/RAPID/TASK1/PROGMOD/KennyWorkingPlan.mod ---
MODULE KennyWorkingPlan
   PERS string workingPlanUUID:="sdvonvskvnwovewn342532nkfloencvosnvqwef12";
    PERS string AP238_WORKINGSTEP_NAME := "";
    PERS string AP238_WORKINGSTEP_UUID := "";
    PERS string AP238_FEATURE_NAME := "";
    PERS string AP238_FEATURE_UUID := "";
    PERS bool ok;
    PERS num startIndex :=134;
    PERS num stopIndex :=140;
      CONST speeddata serge := [ 800, 500, 5000, 1000];



    PROC main()

       !  SetDO IsDone,0;
         MoveAbsJ jHome,v400,z10,PendEff_point\WObj:=A;
        MoveAbsJ jee,v400,z10,PendEff_point\WObj:=A;
        ConfJ\Off;
        ConfL\Off;

       FOR i FROM 1 TO dim(WorkPlan,1) DO

           ok := StrToVal(Workplan{i,1}, startIndex);
           ok := StrToVal(Workplan{i,2}, stopIndex);

                WorkingStep startIndex, stopIndex, Workplan{i,3}, Workplan{i,4}, Workplan{i,5}, Workplan{i,6}, WorkingstepRobtargets, WorkingstepSpeeddatas;

        ENDFOR

        MoveAbsJ jee,v400,z10,PendEff_point\WObj:=A;
        MoveAbsJ jHome,v400,z10,PendEff_point\WObj:=A;
        !SetDO IsDone,0;
    ENDPROC

    PROC WorkingStep(num startpos, num endpos, string workingstepName, string workingstepUUID, string featureName, string featureUUID, robtarget targetList{*}, speeddata speedList{*})

        FOR i FROM startpos TO endpos DO
      !           SetDO IsDone,0;
            AP238_WORKINGSTEP_NAME := workingstepName;
            AP238_WORKINGSTEP_UUID := workingstepUUID;
            AP238_FEATURE_NAME := featureName;
            AP238_FEATURE_UUID := featureUUID;
     !       MoveL targetList{i},v1000,z100,PendEff_point\WObj:=A;
            MoveL Workingsteprobtargets{i}, speedList{i}, z100,PendEff_point\WObj:=A;
     !       SetDO IsDone,1;
            AP238_WORKINGSTEP_NAME := "";
            AP238_WORKINGSTEP_UUID := "";
            AP238_FEATURE_NAME := "";
            AP238_FEATURE_UUID := "";
        ENDFOR

    ENDPROC

ENDMODULE

--- Backups/Rob4/RAPID/TASK1/SYSMOD/WorkObjs.sys ---
MODULE WorkObjs(SYSMODULE)
    TASK PERS wobjdata A:=[FALSE,TRUE,"",[[-982.614,-597.3,290.101],[1,0,0,0]],[[0,0,0],[1,0,0,0]]];
ENDMODULE

